(* Visualisation Lamp_status
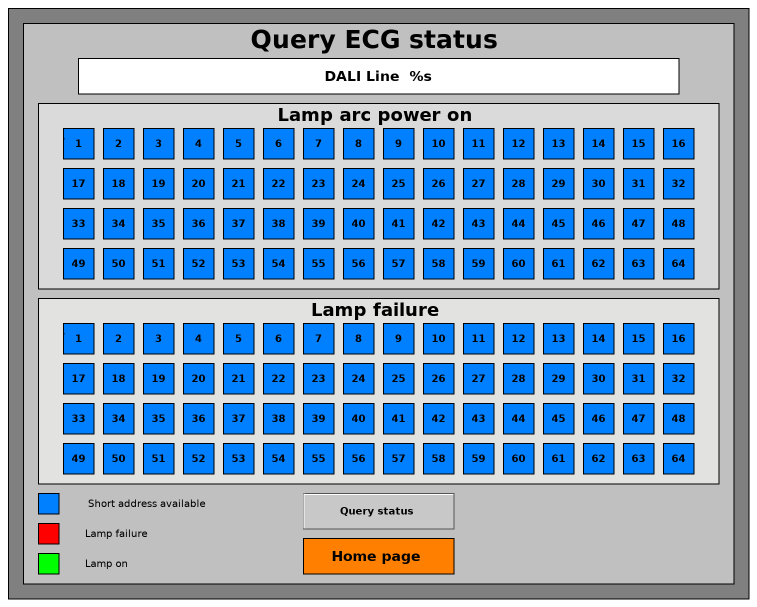
rectangle at (65,35)-(776,596): text "Query ECG status"
rounded rectangle at (345,550)-(496,586): text "Home page"; opens PLC_VISU; tooltip Back to home page
rounded rectangle at (120,70)-(721,106): text "DALI Line  %s"; shows DALI_Config.bDali_Linie; tooltip You can change the DALI Line only on the home page.
rectangle at (80,115)-(761,301): text "Lamp arc power on"
rectangle at (105,140)-(136,171): text "1"; alarm colour if DALI_Config.Kurzadr[1]
rectangle at (105,140)-(136,171): text "1"; invisible if not DALI_Config.Kurzadr[1]; alarm colour if DALI_Config.LampeEin[1]
rectangle at (145,140)-(176,171): text "2"; alarm colour if DALI_Config.Kurzadr[2]
rectangle at (145,140)-(176,171): text "2"; invisible if not DALI_Config.Kurzadr[2]; alarm colour if DALI_Config.LampeEin[2]
rectangle at (185,140)-(216,171): text "3"; alarm colour if DALI_Config.Kurzadr[3]
rectangle at (185,140)-(216,171): text "3"; invisible if not DALI_Config.Kurzadr[3]; alarm colour if DALI_Config.LampeEin[3]
rectangle at (225,140)-(256,171): text "4"; alarm colour if DALI_Config.Kurzadr[4]
rectangle at (225,140)-(256,171): text "4"; invisible if not DALI_Config.Kurzadr[4]; alarm colour if DALI_Config.LampeEin[4]
rectangle at (265,140)-(296,171): text "5"; alarm colour if DALI_Config.Kurzadr[5]
rectangle at (265,140)-(296,171): text "5"; invisible if not DALI_Config.Kurzadr[5]; alarm colour if DALI_Config.LampeEin[5]
rectangle at (305,140)-(336,171): text "6"; alarm colour if DALI_Config.Kurzadr[6]
rectangle at (305,140)-(336,171): text "6"; invisible if not DALI_Config.Kurzadr[6]; alarm colour if DALI_Config.LampeEin[6]
rectangle at (345,140)-(376,171): text "7"; alarm colour if DALI_Config.Kurzadr[7]
rectangle at (345,140)-(376,171): text "7"; invisible if not DALI_Config.Kurzadr[7]; alarm colour if DALI_Config.LampeEin[7]
rectangle at (385,140)-(416,171): text "8"; alarm colour if DALI_Config.Kurzadr[8]
rectangle at (385,140)-(416,171): text "8"; invisible if not DALI_Config.Kurzadr[8]; alarm colour if DALI_Config.LampeEin[8]
rectangle at (425,140)-(456,171): text "9"; alarm colour if DALI_Config.Kurzadr[9]
rectangle at (425,140)-(456,171): text "9"; invisible if not DALI_Config.Kurzadr[9]; alarm colour if DALI_Config.LampeEin[9]
rectangle at (465,140)-(496,171): text "10"; alarm colour if DALI_Config.Kurzadr[10]
rectangle at (465,140)-(496,171): text "10"; invisible if not DALI_Config.Kurzadr[10]; alarm colour if DALI_Config.LampeEin[10]
rectangle at (505,140)-(536,171): text "11"; alarm colour if DALI_Config.Kurzadr[11]
rectangle at (505,140)-(536,171): text "11"; invisible if not DALI_Config.Kurzadr[11]; alarm colour if DALI_Config.LampeEin[11]
rectangle at (545,140)-(576,171): text "12"; alarm colour if DALI_Config.Kurzadr[12]
rectangle at (545,140)-(576,171): text "12"; invisible if not DALI_Config.Kurzadr[12]; alarm colour if DALI_Config.LampeEin[12]
rectangle at (585,140)-(616,171): text "13"; alarm colour if DALI_Config.Kurzadr[13]
rectangle at (585,140)-(616,171): text "13"; invisible if not DALI_Config.Kurzadr[13]; alarm colour if DALI_Config.LampeEin[13]
rectangle at (625,140)-(656,171): text "14"; alarm colour if DALI_Config.Kurzadr[14]
rectangle at (625,140)-(656,171): text "14"; invisible if not DALI_Config.Kurzadr[14]; alarm colour if DALI_Config.LampeEin[14]
rectangle at (665,140)-(696,171): text "15"; alarm colour if DALI_Config.Kurzadr[15]
rectangle at (665,140)-(696,171): text "15"; invisible if not DALI_Config.Kurzadr[15]; alarm colour if DALI_Config.LampeEin[15]
rectangle at (705,140)-(736,171): text "16"; alarm colour if DALI_Config.Kurzadr[16]
rectangle at (705,140)-(736,171): text "16"; invisible if not DALI_Config.Kurzadr[16]; alarm colour if DALI_Config.LampeEin[16]
rectangle at (105,180)-(136,211): text "17"; alarm colour if DALI_Config.Kurzadr[17]
rectangle at (105,180)-(136,211): text "17"; invisible if not DALI_Config.Kurzadr[17]; alarm colour if DALI_Config.LampeEin[17]
rectangle at (185,180)-(216,211): text "19"; alarm colour if DALI_Config.Kurzadr[19]
rectangle at (185,180)-(216,211): text "19"; invisible if not DALI_Config.Kurzadr[19]; alarm colour if DALI_Config.LampeEin[19]
rectangle at (145,180)-(176,211): text "18"; alarm colour if DALI_Config.Kurzadr[18]
rectangle at (145,180)-(176,211): text "18"; invisible if not DALI_Config.Kurzadr[18]; alarm colour if DALI_Config.LampeEin[18]
rectangle at (225,180)-(256,211): text "20"; alarm colour if DALI_Config.Kurzadr[20]
rectangle at (225,180)-(256,211): text "20"; invisible if not DALI_Config.Kurzadr[20]; alarm colour if DALI_Config.LampeEin[20]
rectangle at (265,180)-(296,211): text "21"; alarm colour if DALI_Config.Kurzadr[21]
rectangle at (265,180)-(296,211): text "21"; invisible if not DALI_Config.Kurzadr[21]; alarm colour if DALI_Config.LampeEin[21]
rectangle at (305,180)-(336,211): text "22"; alarm colour if DALI_Config.Kurzadr[22]
rectangle at (305,180)-(336,211): text "22"; invisible if not DALI_Config.Kurzadr[22]; alarm colour if DALI_Config.LampeEin[22]
rectangle at (345,180)-(376,211): text "23"; alarm colour if DALI_Config.Kurzadr[23]
rectangle at (345,180)-(376,211): text "23"; invisible if not DALI_Config.Kurzadr[23]; alarm colour if DALI_Config.LampeEin[23]
rectangle at (385,180)-(416,211): text "24"; alarm colour if DALI_Config.Kurzadr[24]
rectangle at (385,180)-(416,211): text "24"; invisible if not DALI_Config.Kurzadr[24]; alarm colour if DALI_Config.LampeEin[24]
rectangle at (425,180)-(456,211): text "25"; alarm colour if DALI_Config.Kurzadr[25]
rectangle at (425,180)-(456,211): text "25"; invisible if not DALI_Config.Kurzadr[25]; alarm colour if DALI_Config.LampeEin[25]
rectangle at (585,180)-(616,211): text "29"; alarm colour if DALI_Config.Kurzadr[29]
rectangle at (585,180)-(616,211): text "29"; invisible if not DALI_Config.Kurzadr[29]; alarm colour if DALI_Config.LampeEin[29]
rectangle at (545,180)-(576,211): text "28"; alarm colour if DALI_Config.Kurzadr[28]
rectangle at (545,180)-(576,211): text "28"; invisible if not DALI_Config.Kurzadr[28]; alarm colour if DALI_Config.LampeEin[28]
rectangle at (505,180)-(536,211): text "27"; alarm colour if DALI_Config.Kurzadr[27]
rectangle at (505,180)-(536,211): text "27"; invisible if not DALI_Config.Kurzadr[27]; alarm colour if DALI_Config.LampeEin[27]
rectangle at (465,180)-(496,211): text "26"; alarm colour if DALI_Config.Kurzadr[26]
rectangle at (465,180)-(496,211): text "26"; invisible if not DALI_Config.Kurzadr[26]; alarm colour if DALI_Config.LampeEin[26]
rectangle at (625,180)-(656,211): text "30"; alarm colour if DALI_Config.Kurzadr[30]
rectangle at (625,180)-(656,211): text "30"; invisible if not DALI_Config.Kurzadr[30]; alarm colour if DALI_Config.LampeEin[30]
rectangle at (665,180)-(696,211): text "31"; alarm colour if DALI_Config.Kurzadr[31]
rectangle at (665,180)-(696,211): text "31"; invisible if not DALI_Config.Kurzadr[31]; alarm colour if DALI_Config.LampeEin[31]
rectangle at (705,180)-(736,211): text "32"; alarm colour if DALI_Config.Kurzadr[32]
rectangle at (705,180)-(736,211): text "32"; invisible if not DALI_Config.Kurzadr[32]; alarm colour if DALI_Config.LampeEin[32]
rectangle at (105,220)-(136,251): text "33"; alarm colour if DALI_Config.Kurzadr[33]
rectangle at (105,220)-(136,251): text "33"; invisible if not DALI_Config.Kurzadr[33]; alarm colour if DALI_Config.LampeEin[33]
rectangle at (145,220)-(176,251): text "34"; alarm colour if DALI_Config.Kurzadr[34]
rectangle at (145,220)-(176,251): text "34"; invisible if not DALI_Config.Kurzadr[34]; alarm colour if DALI_Config.LampeEin[34]
rectangle at (225,220)-(256,251): text "36"; alarm colour if DALI_Config.Kurzadr[36]
rectangle at (225,220)-(256,251): text "36"; invisible if not DALI_Config.Kurzadr[36]; alarm colour if DALI_Config.LampeEin[36]
rectangle at (305,220)-(336,251): text "38"; alarm colour if DALI_Config.Kurzadr[38]
rectangle at (305,220)-(336,251): text "38"; invisible if not DALI_Config.Kurzadr[38]; alarm colour if DALI_Config.LampeEin[38]
rectangle at (345,220)-(376,251): text "39"; alarm colour if DALI_Config.Kurzadr[39]
rectangle at (345,220)-(376,251): text "39"; invisible if not DALI_Config.Kurzadr[39]; alarm colour if DALI_Config.LampeEin[39]
rectangle at (265,220)-(296,251): text "37"; alarm colour if DALI_Config.Kurzadr[37]
rectangle at (265,220)-(296,251): text "37"; invisible if not DALI_Config.Kurzadr[37]; alarm colour if DALI_Config.LampeEin[37]
rectangle at (185,220)-(216,251): text "35"; alarm colour if DALI_Config.Kurzadr[35]
rectangle at (185,220)-(216,251): text "35"; invisible if not DALI_Config.Kurzadr[35]; alarm colour if DALI_Config.LampeEin[35]
rectangle at (425,220)-(456,251): text "41"; alarm colour if DALI_Config.Kurzadr[41]
rectangle at (425,220)-(456,251): text "41"; invisible if not DALI_Config.Kurzadr[41]; alarm colour if DALI_Config.LampeEin[41]
rectangle at (465,220)-(496,251): text "42"; alarm colour if DALI_Config.Kurzadr[42]
rectangle at (465,220)-(496,251): text "42"; invisible if not DALI_Config.Kurzadr[42]; alarm colour if DALI_Config.LampeEin[42]
rectangle at (385,220)-(416,251): text "40"; alarm colour if DALI_Config.Kurzadr[40]
rectangle at (385,220)-(416,251): text "40"; invisible if not DALI_Config.Kurzadr[40]; alarm colour if DALI_Config.LampeEin[40]
rectangle at (505,220)-(536,251): text "43"; alarm colour if DALI_Config.Kurzadr[43]
rectangle at (505,220)-(536,251): text "43"; invisible if not DALI_Config.Kurzadr[43]; alarm colour if DALI_Config.LampeEin[43]
rectangle at (545,220)-(576,251): text "44"; alarm colour if DALI_Config.Kurzadr[44]
rectangle at (545,220)-(576,251): text "44"; invisible if not DALI_Config.Kurzadr[44]; alarm colour if DALI_Config.LampeEin[44]
rectangle at (585,220)-(616,251): text "45"; alarm colour if DALI_Config.Kurzadr[45]
rectangle at (585,220)-(616,251): text "45"; invisible if not DALI_Config.Kurzadr[45]; alarm colour if DALI_Config.LampeEin[45]
rectangle at (625,220)-(656,251): text "46"; alarm colour if DALI_Config.Kurzadr[46]
rectangle at (625,220)-(656,251): text "46"; invisible if not DALI_Config.Kurzadr[46]; alarm colour if DALI_Config.LampeEin[46]
rectangle at (665,220)-(696,251): text "47"; alarm colour if DALI_Config.Kurzadr[47]
rectangle at (665,220)-(696,251): text "47"; invisible if not DALI_Config.Kurzadr[47]; alarm colour if DALI_Config.LampeEin[47]
rectangle at (705,220)-(736,251): text "48"; alarm colour if DALI_Config.Kurzadr[48]
rectangle at (705,220)-(736,251): text "48"; invisible if not DALI_Config.Kurzadr[48]; alarm colour if DALI_Config.LampeEin[48]
rectangle at (105,260)-(136,291): text "49"; alarm colour if DALI_Config.Kurzadr[49]
rectangle at (105,260)-(136,291): text "49"; invisible if not DALI_Config.Kurzadr[49]; alarm colour if DALI_Config.LampeEin[49]
rectangle at (145,260)-(176,291): text "50"; alarm colour if DALI_Config.Kurzadr[50]
rectangle at (145,260)-(176,291): text "50"; invisible if not DALI_Config.Kurzadr[50]; alarm colour if DALI_Config.LampeEin[50]
rectangle at (185,260)-(216,291): text "51"; alarm colour if DALI_Config.Kurzadr[51]
rectangle at (185,260)-(216,291): text "51"; invisible if not DALI_Config.Kurzadr[51]; alarm colour if DALI_Config.LampeEin[51]
rectangle at (225,260)-(256,291): text "52"; alarm colour if DALI_Config.Kurzadr[52]
rectangle at (225,260)-(256,291): text "52"; invisible if not DALI_Config.Kurzadr[52]; alarm colour if DALI_Config.LampeEin[52]
rectangle at (265,260)-(296,291): text "53"; alarm colour if DALI_Config.Kurzadr[53]
rectangle at (265,260)-(296,291): text "53"; invisible if not DALI_Config.Kurzadr[53]; alarm colour if DALI_Config.LampeEin[53]
rectangle at (305,260)-(336,291): text "54"; alarm colour if DALI_Config.Kurzadr[54]
rectangle at (305,260)-(336,291): text "54"; invisible if not DALI_Config.Kurzadr[54]; alarm colour if DALI_Config.LampeEin[54]
rectangle at (345,260)-(376,291): text "55"; alarm colour if DALI_Config.Kurzadr[55]
rectangle at (345,260)-(376,291): text "55"; invisible if not DALI_Config.Kurzadr[55]; alarm colour if DALI_Config.LampeEin[55]
rectangle at (385,260)-(416,291): text "56"; alarm colour if DALI_Config.Kurzadr[56]
rectangle at (385,260)-(416,291): text "56"; invisible if not DALI_Config.Kurzadr[56]; alarm colour if DALI_Config.LampeEin[56]
rectangle at (425,260)-(456,291): text "57"; alarm colour if DALI_Config.Kurzadr[57]
rectangle at (425,260)-(456,291): text "57"; invisible if not DALI_Config.Kurzadr[57]; alarm colour if DALI_Config.LampeEin[57]
rectangle at (505,260)-(536,291): text "59"; alarm colour if DALI_Config.Kurzadr[59]
rectangle at (505,260)-(536,291): text "59"; invisible if not DALI_Config.Kurzadr[59]; alarm colour if DALI_Config.LampeEin[59]
rectangle at (545,260)-(576,291): text "60"; alarm colour if DALI_Config.Kurzadr[60]
rectangle at (545,260)-(576,291): text "60"; invisible if not DALI_Config.Kurzadr[60]; alarm colour if DALI_Config.LampeEin[60]
rectangle at (585,260)-(616,291): text "61"; alarm colour if DALI_Config.Kurzadr[61]
rectangle at (585,260)-(616,291): text "61"; invisible if not DALI_Config.Kurzadr[61]; alarm colour if DALI_Config.LampeEin[61]
rectangle at (625,260)-(656,291): text "62"; alarm colour if DALI_Config.Kurzadr[62]
rectangle at (625,260)-(656,291): text "62"; invisible if not DALI_Config.Kurzadr[62]; alarm colour if DALI_Config.LampeEin[62]
rectangle at (465,260)-(496,291): text "58"; alarm colour if DALI_Config.Kurzadr[58]
rectangle at (465,260)-(496,291): text "58"; invisible if not DALI_Config.Kurzadr[58]; alarm colour if DALI_Config.LampeEin[58]
rectangle at (665,260)-(696,291): text "63"; alarm colour if DALI_Config.Kurzadr[63]
rectangle at (665,260)-(696,291): text "63"; invisible if not DALI_Config.Kurzadr[63]; alarm colour if DALI_Config.LampeEin[63]
rectangle at (705,260)-(736,291): text "64"; alarm colour if DALI_Config.Kurzadr[64]
rectangle at (705,260)-(736,291): text "64"; invisible if not DALI_Config.Kurzadr[64]; alarm colour if DALI_Config.LampeEin[64]
rectangle at (80,310)-(761,496): text "Lamp failure"
rectangle at (105,335)-(136,366): text "1"; alarm colour if DALI_Config.Kurzadr[1]
rectangle at (105,335)-(136,366): text "1"; invisible if not DALI_Config.Kurzadr[1]; alarm colour if DALI_Config.Lampenausfall[1]
rectangle at (145,335)-(176,366): text "2"; alarm colour if DALI_Config.Kurzadr[2]
rectangle at (145,335)-(176,366): text "2"; invisible if not DALI_Config.Kurzadr[2]; alarm colour if DALI_Config.Lampenausfall[2]
rectangle at (185,335)-(216,366): text "3"; alarm colour if DALI_Config.Kurzadr[3]
rectangle at (185,335)-(216,366): text "3"; invisible if not DALI_Config.Kurzadr[3]; alarm colour if DALI_Config.Lampenausfall[3]
rectangle at (225,335)-(256,366): text "4"; alarm colour if DALI_Config.Kurzadr[4]
rectangle at (225,335)-(256,366): text "4"; invisible if not DALI_Config.Kurzadr[4]; alarm colour if DALI_Config.Lampenausfall[4]
rectangle at (265,335)-(296,366): text "5"; alarm colour if DALI_Config.Kurzadr[5]
rectangle at (265,335)-(296,366): text "5"; invisible if not DALI_Config.Kurzadr[5]; alarm colour if DALI_Config.Lampenausfall[5]
rectangle at (305,335)-(336,366): text "6"; alarm colour if DALI_Config.Kurzadr[6]
rectangle at (305,335)-(336,366): text "6"; invisible if not DALI_Config.Kurzadr[6]; alarm colour if DALI_Config.Lampenausfall[6]
rectangle at (345,335)-(376,366): text "7"; alarm colour if DALI_Config.Kurzadr[7]
rectangle at (345,335)-(376,366): text "7"; invisible if not DALI_Config.Kurzadr[7]; alarm colour if DALI_Config.Lampenausfall[7]
rectangle at (385,335)-(416,366): text "8"; alarm colour if DALI_Config.Kurzadr[8]
rectangle at (385,335)-(416,366): text "8"; invisible if not DALI_Config.Kurzadr[8]; alarm colour if DALI_Config.Lampenausfall[8]
rectangle at (425,335)-(456,366): text "9"; alarm colour if DALI_Config.Kurzadr[9]
rectangle at (425,335)-(456,366): text "9"; invisible if not DALI_Config.Kurzadr[9]; alarm colour if DALI_Config.Lampenausfall[9]
rectangle at (465,335)-(496,366): text "10"; alarm colour if DALI_Config.Kurzadr[10]
rectangle at (465,335)-(496,366): text "10"; invisible if not DALI_Config.Kurzadr[10]; alarm colour if DALI_Config.Lampenausfall[10]
rectangle at (505,335)-(536,366): text "11"; alarm colour if DALI_Config.Kurzadr[11]
rectangle at (505,335)-(536,366): text "11"; invisible if not DALI_Config.Kurzadr[11]; alarm colour if DALI_Config.Lampenausfall[11]
rectangle at (545,335)-(576,366): text "12"; alarm colour if DALI_Config.Kurzadr[12]
rectangle at (545,335)-(576,366): text "12"; invisible if not DALI_Config.Kurzadr[12]; alarm colour if DALI_Config.Lampenausfall[12]
rectangle at (585,335)-(616,366): text "13"; alarm colour if DALI_Config.Kurzadr[13]
rectangle at (585,335)-(616,366): text "13"; invisible if not DALI_Config.Kurzadr[13]; alarm colour if DALI_Config.Lampenausfall[13]
rectangle at (625,335)-(656,366): text "14"; alarm colour if DALI_Config.Kurzadr[14]
rectangle at (625,335)-(656,366): text "14"; invisible if not DALI_Config.Kurzadr[14]; alarm colour if DALI_Config.Lampenausfall[14]
rectangle at (665,335)-(696,366): text "15"; alarm colour if DALI_Config.Kurzadr[15]
rectangle at (665,335)-(696,366): text "15"; invisible if not DALI_Config.Kurzadr[15]; alarm colour if DALI_Config.Lampenausfall[15]
rectangle at (705,335)-(736,366): text "16"; alarm colour if DALI_Config.Kurzadr[16]
rectangle at (705,335)-(736,366): text "16"; invisible if not DALI_Config.Kurzadr[16]; alarm colour if DALI_Config.Lampenausfall[16]
rectangle at (105,375)-(136,406): text "17"; alarm colour if DALI_Config.Kurzadr[17]
rectangle at (105,375)-(136,406): text "17"; invisible if not DALI_Config.Kurzadr[17]; alarm colour if DALI_Config.Lampenausfall[17]
rectangle at (185,375)-(216,406): text "19"; alarm colour if DALI_Config.Kurzadr[19]
rectangle at (185,375)-(216,406): text "19"; invisible if not DALI_Config.Kurzadr[19]; alarm colour if DALI_Config.Lampenausfall[19]
rectangle at (145,375)-(176,406): text "18"; alarm colour if DALI_Config.Kurzadr[18]
rectangle at (145,375)-(176,406): text "18"; invisible if not DALI_Config.Kurzadr[18]; alarm colour if DALI_Config.Lampenausfall[18]
rectangle at (225,375)-(256,406): text "20"; alarm colour if DALI_Config.Kurzadr[20]
rectangle at (225,375)-(256,406): text "20"; invisible if not DALI_Config.Kurzadr[20]; alarm colour if DALI_Config.Lampenausfall[20]
rectangle at (265,375)-(296,406): text "21"; alarm colour if DALI_Config.Kurzadr[21]
rectangle at (265,375)-(296,406): text "21"; invisible if not DALI_Config.Kurzadr[21]; alarm colour if DALI_Config.Lampenausfall[21]
rectangle at (305,375)-(336,406): text "22"; alarm colour if DALI_Config.Kurzadr[22]
rectangle at (305,375)-(336,406): text "22"; invisible if not DALI_Config.Kurzadr[22]; alarm colour if DALI_Config.Lampenausfall[22]
rectangle at (345,375)-(376,406): text "23"; alarm colour if DALI_Config.Kurzadr[23]
rectangle at (345,375)-(376,406): text "23"; invisible if not DALI_Config.Kurzadr[23]; alarm colour if DALI_Config.Lampenausfall[23]
rectangle at (385,375)-(416,406): text "24"; alarm colour if DALI_Config.Kurzadr[24]
rectangle at (385,375)-(416,406): text "24"; invisible if not DALI_Config.Kurzadr[24]; alarm colour if DALI_Config.Lampenausfall[24]
rectangle at (425,375)-(456,406): text "25"; alarm colour if DALI_Config.Kurzadr[25]
rectangle at (425,375)-(456,406): text "25"; invisible if not DALI_Config.Kurzadr[25]; alarm colour if DALI_Config.Lampenausfall[25]
rectangle at (585,375)-(616,406): text "29"; alarm colour if DALI_Config.Kurzadr[29]
rectangle at (585,375)-(616,406): text "29"; invisible if not DALI_Config.Kurzadr[29]; alarm colour if DALI_Config.Lampenausfall[29]
rectangle at (545,375)-(576,406): text "28"; alarm colour if DALI_Config.Kurzadr[28]
rectangle at (545,375)-(576,406): text "28"; invisible if not DALI_Config.Kurzadr[28]; alarm colour if DALI_Config.Lampenausfall[28]
rectangle at (505,375)-(536,406): text "27"; alarm colour if DALI_Config.Kurzadr[27]
rectangle at (505,375)-(536,406): text "27"; invisible if not DALI_Config.Kurzadr[27]; alarm colour if DALI_Config.Lampenausfall[27]
rectangle at (465,375)-(496,406): text "26"; alarm colour if DALI_Config.Kurzadr[26]
rectangle at (465,375)-(496,406): text "26"; invisible if not DALI_Config.Kurzadr[26]; alarm colour if DALI_Config.Lampenausfall[26]
rectangle at (625,375)-(656,406): text "30"; alarm colour if DALI_Config.Kurzadr[30]
rectangle at (625,375)-(656,406): text "30"; invisible if not DALI_Config.Kurzadr[30]; alarm colour if DALI_Config.Lampenausfall[30]
rectangle at (665,375)-(696,406): text "31"; alarm colour if DALI_Config.Kurzadr[31]
rectangle at (665,375)-(696,406): text "31"; invisible if not DALI_Config.Kurzadr[31]; alarm colour if DALI_Config.Lampenausfall[31]
rectangle at (705,375)-(736,406): text "32"; alarm colour if DALI_Config.Kurzadr[32]
rectangle at (705,375)-(736,406): text "32"; invisible if not DALI_Config.Kurzadr[32]; alarm colour if DALI_Config.Lampenausfall[32]
rectangle at (105,415)-(136,446): text "33"; alarm colour if DALI_Config.Kurzadr[33]
rectangle at (105,415)-(136,446): text "33"; invisible if not DALI_Config.Kurzadr[33]; alarm colour if DALI_Config.Lampenausfall[33]
rectangle at (145,415)-(176,446): text "34"; alarm colour if DALI_Config.Kurzadr[34]
rectangle at (145,415)-(176,446): text "34"; invisible if not DALI_Config.Kurzadr[34]; alarm colour if DALI_Config.Lampenausfall[34]
rectangle at (225,415)-(256,446): text "36"; alarm colour if DALI_Config.Kurzadr[36]
rectangle at (225,415)-(256,446): text "36"; invisible if not DALI_Config.Kurzadr[36]; alarm colour if DALI_Config.Lampenausfall[36]
rectangle at (305,415)-(336,446): text "38"; alarm colour if DALI_Config.Kurzadr[38]
rectangle at (305,415)-(336,446): text "38"; invisible if not DALI_Config.Kurzadr[38]; alarm colour if DALI_Config.Lampenausfall[38]
rectangle at (345,415)-(376,446): text "39"; alarm colour if DALI_Config.Kurzadr[39]
rectangle at (345,415)-(376,446): text "39"; invisible if not DALI_Config.Kurzadr[39]; alarm colour if DALI_Config.Lampenausfall[39]
rectangle at (265,415)-(296,446): text "37"; alarm colour if DALI_Config.Kurzadr[37]
rectangle at (265,415)-(296,446): text "37"; invisible if not DALI_Config.Kurzadr[37]; alarm colour if DALI_Config.Lampenausfall[37]
rectangle at (185,415)-(216,446): text "35"; alarm colour if DALI_Config.Kurzadr[35]
rectangle at (185,415)-(216,446): text "35"; invisible if not DALI_Config.Kurzadr[35]; alarm colour if DALI_Config.Lampenausfall[35]
rectangle at (425,415)-(456,446): text "41"; alarm colour if DALI_Config.Kurzadr[41]
rectangle at (425,415)-(456,446): text "41"; invisible if not DALI_Config.Kurzadr[41]; alarm colour if DALI_Config.Lampenausfall[41]
rectangle at (465,415)-(496,446): text "42"; alarm colour if DALI_Config.Kurzadr[42]
rectangle at (465,415)-(496,446): text "42"; invisible if not DALI_Config.Kurzadr[42]; alarm colour if DALI_Config.Lampenausfall[42]
rectangle at (385,415)-(416,446): text "40"; alarm colour if DALI_Config.Kurzadr[40]
rectangle at (385,415)-(416,446): text "40"; invisible if not DALI_Config.Kurzadr[40]; alarm colour if DALI_Config.Lampenausfall[40]
rectangle at (505,415)-(536,446): text "43"; alarm colour if DALI_Config.Kurzadr[43]
rectangle at (505,415)-(536,446): text "43"; invisible if not DALI_Config.Kurzadr[43]; alarm colour if DALI_Config.Lampenausfall[43]
rectangle at (545,415)-(576,446): text "44"; alarm colour if DALI_Config.Kurzadr[44]
rectangle at (545,415)-(576,446): text "44"; invisible if not DALI_Config.Kurzadr[44]; alarm colour if DALI_Config.Lampenausfall[44]
rectangle at (585,415)-(616,446): text "45"; alarm colour if DALI_Config.Kurzadr[45]
rectangle at (585,415)-(616,446): text "45"; invisible if not DALI_Config.Kurzadr[45]; alarm colour if DALI_Config.Lampenausfall[45]
rectangle at (625,415)-(656,446): text "46"; alarm colour if DALI_Config.Kurzadr[46]
rectangle at (625,415)-(656,446): text "46"; invisible if not DALI_Config.Kurzadr[46]; alarm colour if DALI_Config.Lampenausfall[46]
rectangle at (665,415)-(696,446): text "47"; alarm colour if DALI_Config.Kurzadr[47]
rectangle at (665,415)-(696,446): text "47"; invisible if not DALI_Config.Kurzadr[47]; alarm colour if DALI_Config.Lampenausfall[47]
rectangle at (705,415)-(736,446): text "48"; alarm colour if DALI_Config.Kurzadr[48]
rectangle at (705,415)-(736,446): text "48"; invisible if not DALI_Config.Kurzadr[48]; alarm colour if DALI_Config.Lampenausfall[48]
rectangle at (105,455)-(136,486): text "49"; alarm colour if DALI_Config.Kurzadr[49]
rectangle at (105,455)-(136,486): text "49"; invisible if not DALI_Config.Kurzadr[49]; alarm colour if DALI_Config.Lampenausfall[49]
rectangle at (145,455)-(176,486): text "50"; alarm colour if DALI_Config.Kurzadr[50]
rectangle at (145,455)-(176,486): text "50"; invisible if not DALI_Config.Kurzadr[50]; alarm colour if DALI_Config.Lampenausfall[50]
rectangle at (185,455)-(216,486): text "51"; alarm colour if DALI_Config.Kurzadr[51]
rectangle at (185,455)-(216,486): text "51"; invisible if not DALI_Config.Kurzadr[51]; alarm colour if DALI_Config.Lampenausfall[51]
rectangle at (225,455)-(256,486): text "52"; alarm colour if DALI_Config.Kurzadr[52]
rectangle at (225,455)-(256,486): text "52"; invisible if not DALI_Config.Kurzadr[52]; alarm colour if DALI_Config.Lampenausfall[52]
rectangle at (265,455)-(296,486): text "53"; alarm colour if DALI_Config.Kurzadr[53]
rectangle at (265,455)-(296,486): text "53"; invisible if not DALI_Config.Kurzadr[53]; alarm colour if DALI_Config.Lampenausfall[53]
rectangle at (305,455)-(336,486): text "54"; alarm colour if DALI_Config.Kurzadr[54]
rectangle at (305,455)-(336,486): text "54"; invisible if not DALI_Config.Kurzadr[54]; alarm colour if DALI_Config.Lampenausfall[54]
rectangle at (345,455)-(376,486): text "55"; alarm colour if DALI_Config.Kurzadr[55]
rectangle at (345,455)-(376,486): text "55"; invisible if not DALI_Config.Kurzadr[55]; alarm colour if DALI_Config.Lampenausfall[55]
rectangle at (385,455)-(416,486): text "56"; alarm colour if DALI_Config.Kurzadr[56]
rectangle at (385,455)-(416,486): text "56"; invisible if not DALI_Config.Kurzadr[56]; alarm colour if DALI_Config.Lampenausfall[56]
rectangle at (425,455)-(456,486): text "57"; alarm colour if DALI_Config.Kurzadr[57]
rectangle at (425,455)-(456,486): text "57"; invisible if not DALI_Config.Kurzadr[57]; alarm colour if DALI_Config.Lampenausfall[57]
rectangle at (505,455)-(536,486): text "59"; alarm colour if DALI_Config.Kurzadr[59]
rectangle at (505,455)-(536,486): text "59"; invisible if not DALI_Config.Kurzadr[59]; alarm colour if DALI_Config.Lampenausfall[59]
rectangle at (545,455)-(576,486): text "60"; alarm colour if DALI_Config.Kurzadr[60]
rectangle at (545,455)-(576,486): text "60"; invisible if not DALI_Config.Kurzadr[60]; alarm colour if DALI_Config.Lampenausfall[60]
rectangle at (585,455)-(616,486): text "61"; alarm colour if DALI_Config.Kurzadr[61]
rectangle at (585,455)-(616,486): text "61"; invisible if not DALI_Config.Kurzadr[61]; alarm colour if DALI_Config.Lampenausfall[61]
rectangle at (625,455)-(656,486): text "62"; alarm colour if DALI_Config.Kurzadr[62]
rectangle at (625,455)-(656,486): text "62"; invisible if not DALI_Config.Kurzadr[62]; alarm colour if DALI_Config.Lampenausfall[62]
rectangle at (465,455)-(496,486): text "58"; alarm colour if DALI_Config.Kurzadr[58]
rectangle at (465,455)-(496,486): text "58"; invisible if not DALI_Config.Kurzadr[58]; alarm colour if DALI_Config.Lampenausfall[58]
rectangle at (665,455)-(696,486): text "63"; alarm colour if DALI_Config.Kurzadr[63]
rectangle at (665,455)-(696,486): text "63"; invisible if not DALI_Config.Kurzadr[63]; alarm colour if DALI_Config.Lampenausfall[63]
rectangle at (705,455)-(736,486): text "64"; alarm colour if DALI_Config.Kurzadr[64]
rectangle at (705,455)-(736,486): text "64"; invisible if not DALI_Config.Kurzadr[64]; alarm colour if DALI_Config.Lampenausfall[64]
button at (345,505)-(496,541): text "Query status"; taps DALI_Config.Status; tooltip If you click the button "Query Status", you will get the status "Lamp failure" and "Lamp arc power on" from the ECG.
rectangle at (110,505)-(271,526): text "Short address available"
rectangle at (125,535)-(256,556): text "Lamp failure"
rectangle at (125,565)-(196,586): text "Lamp on"
6 more shapes without text or variables
*)

(* Visualisation lux
rectangle at (915,525)-(1011,546): text "Zpet"; opens PLC_VISU; tooltip Back to home page
1 elements of other kinds (tables, trends, ...) not read
*)

(* Visualisation PLC_VISU
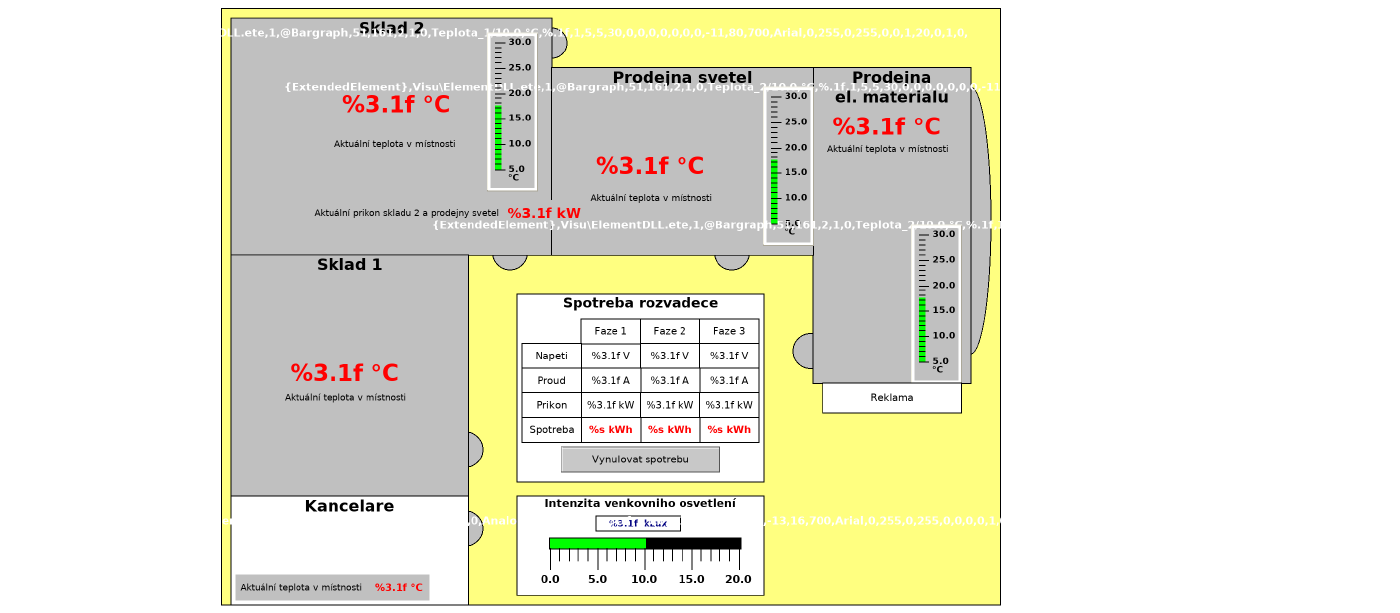
ellipse at (740,80)-(781,351): opens CasProg
ellipse at (580,330)-(616,366): alarm colour if .KA13; taps .TL10s; tooltip Dlouhý stisk zapne svìtlo. (cca 1s)
rectangle at (600,60)-(761,381): text "Prodejna"; opens prodej_materialu
ellipse at (500,230)-(536,266): alarm colour if .KA13; taps .TL10s; tooltip Dlouhý stisk zapne svìtlo. (cca 1s)
ellipse at (275,230)-(311,266): alarm colour if .KA16; taps .TL05s; tooltip Dlouhý stisk zapne svìtlo. (cca 1s)
ellipse at (320,20)-(351,51): alarm colour if .KA15; taps .TL06s; tooltip Dlouhý stisk zapne svìtlo. (cca 1s)
rectangle at (10,10)-(336,251): text "Sklad 2"; opens DALI_cfg
rectangle at (10,250)-(251,496): text "Sklad 1"; opens DALI_cfg
rectangle at (335,60)-(601,251): text "Prodejna svetel"; opens prodej_svetel
rectangle at (10,495)-(251,606): text "Kancelare"
rectangle at (60,380)-(201,411): text "Aktuální teplota v místnosti"
rectangle at (70,350)-(181,391): text "%3.1f °C"; shows .Teplota_3/10.0
rectangle at (110,125)-(251,151): text "Aktuální teplota v místnosti"
rectangle at (120,70)-(236,126): text "%3.1f °C"; shows .Teplota_1/10.0
rectangle at (380,130)-(491,191): text "%3.1f °C"; shows .Teplota_2/10.0
rectangle at (370,180)-(506,206): text "Aktuální teplota v místnosti"
rectangle at (15,575)-(151,601): text "Aktuální teplota v místnosti"
rectangle at (150,575)-(211,601): text "%3.1f °C"; shows .Teplota_4/10.0
rounded rectangle at (300,290)-(551,481): text "Spotreba rozvadece"
rectangle at (365,340)-(426,366): text "%3.1f V"; shows TriFaze.arNapeti[1]
rectangle at (365,315)-(426,341): text "Faze 1"
rectangle at (425,315)-(486,341): text "Faze 2"
rectangle at (485,315)-(546,341): text "Faze 3"
rectangle at (425,340)-(486,366): text "%3.1f V"; shows TriFaze.arNapeti[2]
rectangle at (485,340)-(546,366): text "%3.1f V"; shows TriFaze.arNapeti[3]
rectangle at (485,365)-(546,391): text "%3.1f A"; shows TriFaze.arProud[3]
rectangle at (425,365)-(486,391): text "%3.1f A"; shows TriFaze.arProud[2]
rectangle at (365,365)-(426,391): text "%3.1f A"; shows TriFaze.arProud[1]
rectangle at (365,390)-(426,416): text "%3.1f kW"; shows TriFaze.arVykon[1]
rectangle at (425,390)-(486,416): text "%3.1f kW"; shows TriFaze.arVykon[2]
rectangle at (485,390)-(546,416): text "%3.1f kW"; shows TriFaze.arVykon[3]
rectangle at (485,415)-(546,441): text "%s kWh"; shows TriFaze.adwSpotreba[3]
rectangle at (425,415)-(486,441): text "%s kWh"; shows TriFaze.adwSpotreba[2]
rectangle at (365,415)-(426,441): text "%s kWh"; shows TriFaze.adwSpotreba[1]
button at (345,445)-(506,471): text "Vynulovat spotrebu"; taps TriFaze.SmazL1
rounded rectangle at (300,495)-(551,596): text "Intenzita venkovniho osvetlení"; opens lux
rectangle at (380,515)-(466,531): text "%3.1f  kLux"; shows .Analog_1/3276.4*2
rectangle at (305,340)-(366,366): text "Napeti"
rectangle at (305,365)-(366,391): text "Proud"
rectangle at (305,390)-(366,416): text "Prikon"
rectangle at (305,415)-(366,441): text "Spotreba"
rectangle at (90,195)-(301,221): text "Aktuální prikon skladu 2 a prodejny svetel"
rectangle at (295,195)-(361,221): text "%3.1f kW"; shows TriFaze.arVykon[1]+TriFaze.arVykon[2]+TriFaze.arVykon[3]
group at (320,520)-(541,621)
  rectangle at (0,0)-(1,1): text "{ExtendedElement},Visu\ElementDLL.ete,1,@Bargraph,221,111,0,0,0,Analog_1/3276.4*2,,%.1f,1,5,0,20,0,0,0,0,0,0,0,-13,16,700,Arial,0,255,0,255,0,0,0,0,1,0,0,"
  rectangle at (14,19)-(111,29): alarm colour if (Analog_1/3276.4*2) < 0; right ((Analog_1/3276.4*2 * 1.0) - 10)  * 9.6
  rectangle at (2,53)-(26,103): text "0.0"
  rectangle at (50,53)-(74,103): text "5.0"
  rectangle at (93,53)-(126,103): text "10.0"
  rectangle at (141,53)-(174,103): text "15.0"
  rectangle at (189,53)-(222,103): text "20.0"
group at (550,80)-(601,241)
  rectangle at (0,0)-(1,1): text "{ExtendedElement},Visu\ElementDLL.ete,1,@Bargraph,51,161,2,1,0,Teplota_2/10.0,°C,%.1f,1,5,5,30,0,0,0,0,0,0,0,-11,80,700,Arial,0,255,0,255,0,0,1,25,0,1,0,"
  rectangle at (8,74)-(14,139): alarm colour if (Teplota_2/10.0) > 25; top ((Teplota_2/10.0 * 1.0) - 17.5)  * -5.2
  rectangle at (20,129)-(47,148): text "5.0"
  rectangle at (20,103)-(47,122): text "10.0"
  rectangle at (20,77)-(47,96): text "15.0"
  rectangle at (20,52)-(47,71): text "20.0"
  rectangle at (20,26)-(47,45): text "25.0"
  rectangle at (20,0)-(47,19): text "30.0"
  rectangle at (15,140)-(39,154): text "°C"
group at (270,25)-(321,186)
  rectangle at (0,0)-(1,1): text "{ExtendedElement},Visu\ElementDLL.ete,1,@Bargraph,51,161,2,1,0,Teplota_1/10.0,°C,%.1f,1,5,5,30,0,0,0,0,0,0,0,-11,80,700,Arial,0,255,0,255,0,0,1,20,0,1,0,"
  rectangle at (8,74)-(14,139): alarm colour if (Teplota_1/10.0) > 20; top ((Teplota_1/10.0 * 1.0) - 17.5)  * -5.2
  rectangle at (20,129)-(47,148): text "5.0"
  rectangle at (20,103)-(47,122): text "10.0"
  rectangle at (20,77)-(47,96): text "15.0"
  rectangle at (20,52)-(47,71): text "20.0"
  rectangle at (20,26)-(47,45): text "25.0"
  rectangle at (20,0)-(47,19): text "30.0"
  rectangle at (15,140)-(39,154): text "°C"
group at (700,220)-(751,381)
  rectangle at (0,0)-(1,1): text "{ExtendedElement},Visu\ElementDLL.ete,1,@Bargraph,51,161,2,1,0,Teplota_2/10.0,°C,%.1f,1,5,5,30,0,0,0,0,0,0,0,-11,80,700,Arial,0,255,0,255,0,0,1,25,0,1,0,"
  rectangle at (8,74)-(14,139): alarm colour if (Teplota_2/10.0) > 25; top ((Teplota_2/10.0 * 1.0) - 17.5)  * -5.2
  rectangle at (20,129)-(47,148): text "5.0"
  rectangle at (20,103)-(47,122): text "10.0"
  rectangle at (20,77)-(47,96): text "15.0"
  rectangle at (20,52)-(47,71): text "20.0"
  rectangle at (20,26)-(47,45): text "25.0"
  rectangle at (20,0)-(47,19): text "30.0"
  rectangle at (15,140)-(39,154): text "°C"
rectangle at (620,90)-(731,151): text "%3.1f °C"
rectangle at (610,130)-(746,156): text "Aktuální teplota v místnosti"
rectangle at (620,80)-(741,101): text "el. materialu"; opens prodej_materialu
rectangle at (610,380)-(751,411): text "Reklama"; opens CasProg
127 more shapes without text or variables
*)

(* Visualisation prodej_materialu
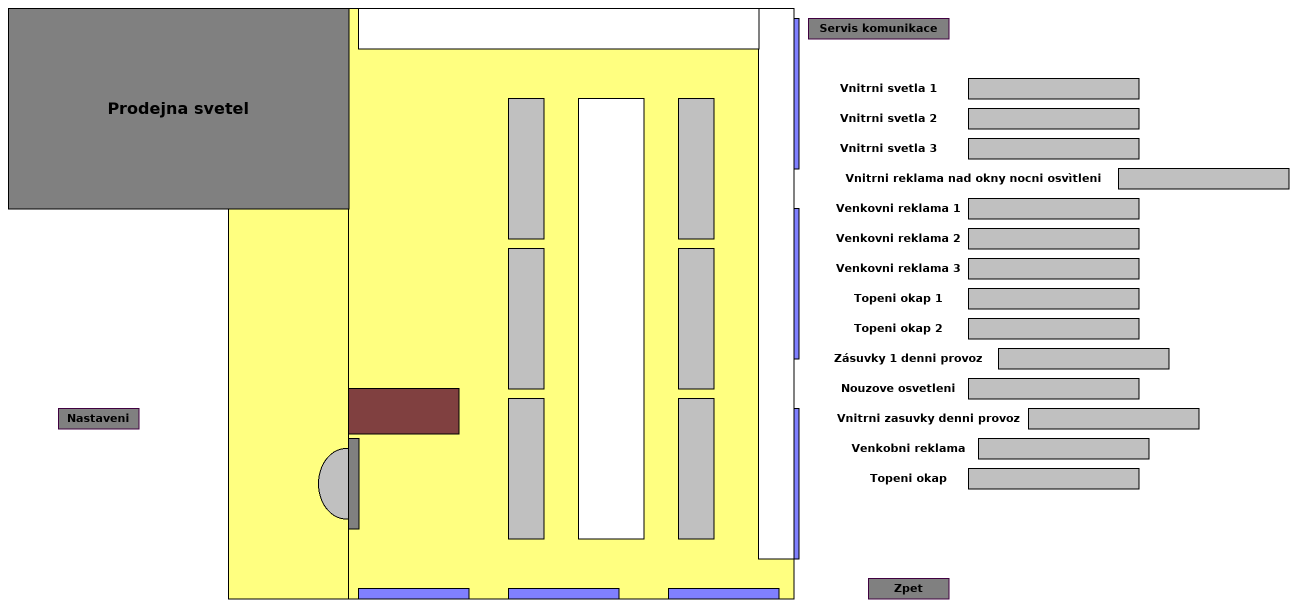
ellipse at (310,440)-(366,511): alarm colour if OUTSvetloNadVchodem; taps INSvetloNadVchodem; tooltip Dlouhý stisk zapne svìtlo. (cca 1s)
rectangle at (860,570)-(941,591): text "Zpet"; opens PLC_VISU; tooltip Back to home page
rectangle at (670,90)-(706,231): tooltip Kliknutím zapínáte a vypínáte svìtla DALI
rectangle at (670,240)-(706,381): tooltip Kliknutím zapínáte a vypínáte svìtla DALI
rectangle at (670,390)-(706,531): tooltip Kliknutím zapínáte a vypínáte svìtla DALI
rectangle at (500,90)-(536,231): tooltip Kliknutím zapínáte a vypínáte svìtla DALI
rectangle at (500,240)-(536,381): tooltip Kliknutím zapínáte a vypínáte svìtla DALI
rectangle at (500,390)-(536,531): tooltip Kliknutím zapínáte a vypínáte svìtla DALI
rectangle at (0,0)-(341,201): text "Prodejna svetel"; opens prodej_svetel
rectangle at (750,0)-(786,551): tooltip Kliknutím zapínáte a vypínáte svìtla DALI
rectangle at (570,90)-(636,531): tooltip Kliknutím zapínáte a vypínáte svìtla DALI
rectangle at (350,0)-(751,41): tooltip Kliknutím zapínáte a vypínáte svìtla DALI
rectangle at (800,10)-(941,31): text "Servis komunikace"; opens ServisNovaProdejna; tooltip Back to home page
rectangle at (960,70)-(1131,91): alarm colour if OUTVnitrniSvetla1; taps INVnitrniSvetla1; tooltip Kliknutím zapínáte a vypínáte svìtla DALI
rectangle at (810,70)-(951,91): text "Vnitrni svetla 1"
rectangle at (810,100)-(951,121): text "Vnitrni svetla 2"
rectangle at (810,130)-(951,151): text "Vnitrni svetla 3"
rectangle at (810,160)-(1121,181): text "Vnitrni reklama nad okny nocni osvìtleni"
rectangle at (820,190)-(961,211): text "Venkovni reklama 1"
rectangle at (820,220)-(961,241): text "Venkovni reklama 2"
rectangle at (820,250)-(961,271): text "Venkovni reklama 3"
rectangle at (820,280)-(961,301): text "Topeni okap 1"
rectangle at (820,310)-(961,331): text "Topeni okap 2"
rectangle at (820,340)-(981,361): text "Zásuvky 1 denni provoz"
rectangle at (820,370)-(961,391): text "Nouzove osvetleni"
rectangle at (820,400)-(1021,421): text "Vnitrni zasuvky denni provoz"
rectangle at (830,430)-(971,451): text "Venkobni reklama"
rectangle at (830,460)-(971,481): text "Topeni okap"
rectangle at (960,100)-(1131,121): alarm colour if OUTVnitrniSvetla2; taps INVnitrniSvetla2; tooltip Kliknutím zapínáte a vypínáte svìtla DALI
rectangle at (960,130)-(1131,151): alarm colour if OUTVnitrniSvetla3; taps INVnitrniSvetla3; tooltip Kliknutím zapínáte a vypínáte svìtla DALI
rectangle at (1110,160)-(1281,181): alarm colour if OUTVnitrniReklama; taps INVnitrniReklama; tooltip Kliknutím zapínáte a vypínáte svìtla DALI
rectangle at (960,190)-(1131,211): alarm colour if OUTVenkovniReklama1; taps INVenkovniReklama; tooltip Kliknutím zapínáte a vypínáte svìtla DALI
rectangle at (960,220)-(1131,241): alarm colour if OUTVenkovniReklama2; taps INVenkovniReklama; tooltip Kliknutím zapínáte a vypínáte svìtla DALI
rectangle at (960,250)-(1131,271): alarm colour if OUTVenkovniReklama3; taps INVenkovniReklama; tooltip Kliknutím zapínáte a vypínáte svìtla DALI
rectangle at (960,280)-(1131,301): alarm colour if OUTTopeniOkap1; taps INTopeniOkap; tooltip Kliknutím zapínáte a vypínáte svìtla DALI
rectangle at (960,310)-(1131,331): alarm colour if OUTTopeniOkap2; taps INTopeniOkap; tooltip Kliknutím zapínáte a vypínáte svìtla DALI
rectangle at (960,460)-(1131,481): alarm colour if OUTTopeniOkap; taps INTopeniOkap; tooltip Kliknutím zapínáte a vypínáte svìtla DALI
rectangle at (990,340)-(1161,361): alarm colour if OUTZasuvky1; tooltip Kliknutím zapínáte a vypínáte svìtla DALI
rectangle at (960,370)-(1131,391): alarm colour if OUTNouzoveOsvetleni; tooltip Kliknutím zapínáte a vypínáte svìtla DALI
rectangle at (1020,400)-(1191,421): alarm colour if OUTVnitrniZasuvkyDenniProvoz; taps INVnitrniZasuvkyDenniProvoz; tooltip Kliknutím zapínáte a vypínáte svìtla DALI
rectangle at (970,430)-(1141,451): alarm colour if OUTVnitrniReklama; taps INVnitrniReklama; tooltip Kliknutím zapínáte a vypínáte svìtla DALI
rectangle at (50,400)-(131,421): text "Nastaveni"; opens prodej_materialu_nastaveni; tooltip Back to home page
10 more shapes without text or variables
*)

(* Visualisation prodej_materialu_nastaveni
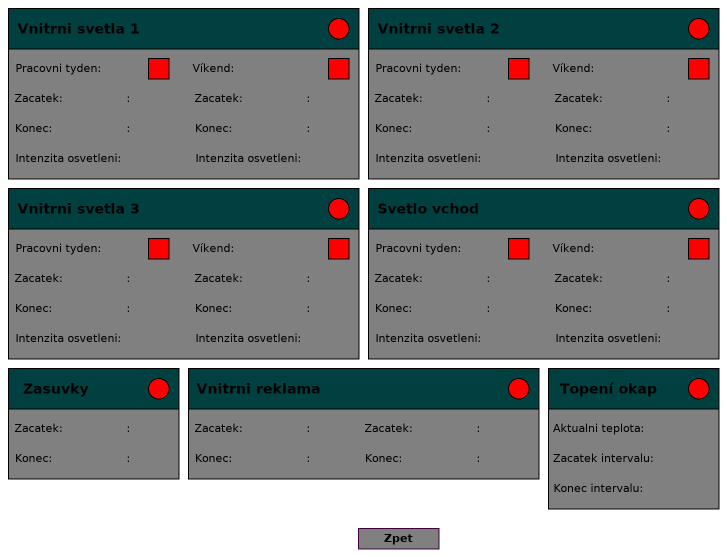
rectangle at (10,10)-(151,51): text "Vnitrni svetla 1"
ellipse at (330,20)-(351,41): alarm colour if ProdejnaMaterialu.PRGVnitrniSvetla1; toggles ProdejnaMaterialu.PRGVnitrniSvetla1
rectangle at (10,90)-(71,111): text "Zacatek:"
rectangle at (10,120)-(61,141): text "Konec:"
rectangle at (120,90)-(141,111): text ":"
rectangle at (120,120)-(141,141): text ":"
rectangle at (10,370)-(111,411): text "Zasuvky"
ellipse at (150,380)-(171,401): alarm colour if ProdejnaMaterialu.PRGVnitrniZasuvkyDenniProvoz; toggles ProdejnaMaterialu.PRGVnitrniZasuvkyDenniProvoz
rectangle at (10,420)-(71,441): text "Zacatek:"
rectangle at (10,450)-(61,471): text "Konec:"
rectangle at (120,420)-(141,441): text ":"
rectangle at (120,450)-(141,471): text ":"
rectangle at (370,190)-(491,231): text "Svetlo vchod"
ellipse at (690,200)-(711,221): alarm colour if ProdejnaMaterialu.PRGSvetloNadVchodem; toggles ProdejnaMaterialu.PRGSvetloNadVchodem
rectangle at (370,270)-(431,291): text "Zacatek:"
rectangle at (370,300)-(421,321): text "Konec:"
rectangle at (480,270)-(501,291): text ":"
rectangle at (480,300)-(501,321): text ":"
rectangle at (190,370)-(331,411): text "Vnitrni reklama"
ellipse at (510,380)-(531,401): alarm colour if ProdejnaMaterialu.PRGVnitrniReklama; toggles ProdejnaMaterialu.PRGVnitrniReklama
rectangle at (190,420)-(251,441): text "Zacatek:"
rectangle at (190,450)-(241,471): text "Konec:"
rectangle at (300,420)-(321,441): text ":"
rectangle at (300,450)-(321,471): text ":"
rectangle at (360,420)-(421,441): text "Zacatek:"
rectangle at (360,450)-(411,471): text "Konec:"
rectangle at (470,420)-(491,441): text ":"
rectangle at (470,450)-(491,471): text ":"
rectangle at (550,370)-(671,411): text "Topení okap"
ellipse at (690,380)-(711,401): alarm colour if INTopeniOkap
rectangle at (550,420)-(651,441): text "Aktualni teplota:"
rectangle at (550,450)-(661,471): text "Zacatek intervalu:"; tooltip Nejnižší teplota.
rectangle at (550,480)-(651,501): text "Konec intervalu:"; tooltip Nevyšší teplota.
rectangle at (10,150)-(131,171): text "Intenzita osvetleni:"
rectangle at (370,330)-(491,351): text "Intenzita osvetleni:"
rectangle at (370,240)-(471,261): text "Pracovni tyden:"
rectangle at (510,240)-(531,261): alarm colour if ProdejnaMaterialu.xSvetloNadVchodemPracTyden; toggles ProdejnaMaterialu.xSvetloNadVchodemPracTyden
rectangle at (550,270)-(611,291): text "Zacatek:"
rectangle at (550,300)-(601,321): text "Konec:"
rectangle at (660,270)-(681,291): text ":"
rectangle at (660,300)-(681,321): text ":"
rectangle at (550,330)-(671,351): text "Intenzita osvetleni:"
rectangle at (550,240)-(601,261): text "Víkend:"
rectangle at (690,240)-(711,261): alarm colour if ProdejnaMaterialu.xSvetloNadVchodemVikend; toggles ProdejnaMaterialu.xSvetloNadVchodemVikend
rectangle at (10,60)-(111,81): text "Pracovni tyden:"
rectangle at (150,60)-(171,81): alarm colour if ProdejnaMaterialu.xVnitrniSvetla1PracDen; toggles ProdejnaMaterialu.xVnitrniSvetla1PracDen
rectangle at (190,60)-(241,81): text "Víkend:"
rectangle at (330,60)-(351,81): alarm colour if ProdejnaMaterialu.xVnitrniSvetla1Vikend; toggles ProdejnaMaterialu.xVnitrniSvetla1Vikend
rectangle at (190,90)-(251,111): text "Zacatek:"
rectangle at (190,120)-(241,141): text "Konec:"
rectangle at (300,90)-(321,111): text ":"
rectangle at (300,120)-(321,141): text ":"
rectangle at (190,150)-(311,171): text "Intenzita osvetleni:"
rectangle at (370,10)-(511,51): text "Vnitrni svetla 2"
ellipse at (690,20)-(711,41): alarm colour if ProdejnaMaterialu.PRGVnitrniSvetla2; toggles ProdejnaMaterialu.PRGVnitrniSvetla2
rectangle at (370,90)-(431,111): text "Zacatek:"
rectangle at (370,120)-(421,141): text "Konec:"
rectangle at (480,90)-(501,111): text ":"
rectangle at (480,120)-(501,141): text ":"
rectangle at (370,150)-(491,171): text "Intenzita osvetleni:"
rectangle at (370,60)-(471,81): text "Pracovni tyden:"
rectangle at (510,60)-(531,81): alarm colour if ProdejnaMaterialu.xVnitrniSvetla2PracDen; toggles ProdejnaMaterialu.xVnitrniSvetla2PracDen
rectangle at (550,60)-(601,81): text "Víkend:"
rectangle at (690,60)-(711,81): alarm colour if ProdejnaMaterialu.xVnitrniSvetla2Vikend; toggles ProdejnaMaterialu.xVnitrniSvetla2Vikend
rectangle at (550,90)-(611,111): text "Zacatek:"
rectangle at (550,120)-(601,141): text "Konec:"
rectangle at (660,90)-(681,111): text ":"
rectangle at (660,120)-(681,141): text ":"
rectangle at (550,150)-(671,171): text "Intenzita osvetleni:"
rectangle at (10,190)-(151,231): text "Vnitrni svetla 3"
ellipse at (330,200)-(351,221): alarm colour if ProdejnaMaterialu.PRGVnitrniSvetla3; toggles ProdejnaMaterialu.PRGVnitrniSvetla3
rectangle at (10,270)-(71,291): text "Zacatek:"
rectangle at (10,300)-(61,321): text "Konec:"
rectangle at (120,270)-(141,291): text ":"
rectangle at (120,300)-(141,321): text ":"
rectangle at (10,330)-(131,351): text "Intenzita osvetleni:"
rectangle at (10,240)-(111,261): text "Pracovni tyden:"
rectangle at (150,240)-(171,261): alarm colour if ProdejnaMaterialu.xVnitrniSvetla3PracDen; toggles ProdejnaMaterialu.xVnitrniSvetla3PracDen
rectangle at (190,240)-(241,261): text "Víkend:"
rectangle at (330,240)-(351,261): alarm colour if ProdejnaMaterialu.xVnitrniSvetla3Vikend; toggles ProdejnaMaterialu.xVnitrniSvetla3Vikend
rectangle at (190,270)-(251,291): text "Zacatek:"
rectangle at (190,300)-(241,321): text "Konec:"
rectangle at (300,270)-(321,291): text ":"
rectangle at (300,300)-(321,321): text ":"
rectangle at (190,330)-(311,351): text "Intenzita osvetleni:"
rectangle at (360,530)-(441,551): text "Zpet"; opens prodej_materialu; tooltip Back to home page
14 more shapes without text or variables
55 elements of other kinds (tables, trends, ...) not read
*)

(* Visualisation prodej_svetel
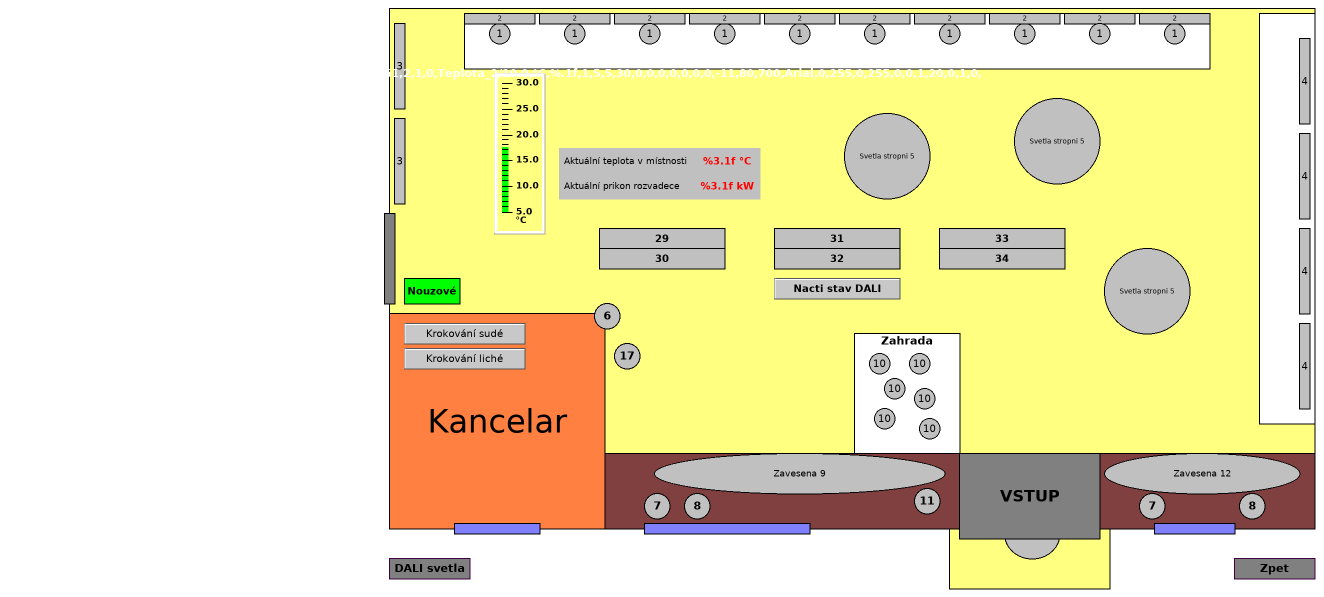
rounded rectangle at (485,345)-(591,476): text "Zahrada"
ellipse at (635,520)-(691,571): alarm colour if .KA13; taps .TL10s; tooltip Dlouhý stisk zapne svìtlo. (cca 1s)
rectangle at (25,130)-(36,216): text "3"; alarm colour if .KA03
rectangle at (35,290)-(91,316): text "Nouzové"; alarm colour if .KA20
rectangle at (20,325)-(236,541): text "Kancelar"
rectangle at (865,570)-(946,591): text "Zpet"; opens PLC_VISU; tooltip Back to home page
ellipse at (315,505)-(341,531): text "8"; alarm colour if .ka08
ellipse at (735,465)-(931,506): text "Zavesena 12"; alarm colour if .KA12
rectangle at (930,50)-(941,136): text "4"; alarm colour if .KA04
ellipse at (500,365)-(521,386): text "10"; alarm colour if .KA10
ellipse at (285,465)-(576,506): text "Zavesena 9"; alarm colour if .KA09
rectangle at (590,465)-(731,551): text "VSTUP"
rectangle at (325,160)-(391,186): text "%3.1f °C"; shows .Teplota_2/10.0
rectangle at (190,160)-(326,186): text "Aktuální teplota v místnosti"
ellipse at (120,35)-(141,56): text "1"; alarm colour if .KA01; taps .TL10s; tooltip Klinutím zapínáte žárovky na deskách
rectangle at (95,25)-(166,36): text "2"; alarm colour if .KA02
ellipse at (275,505)-(301,531): text "7"; alarm colour if .ka07
ellipse at (870,505)-(896,531): text "8"; alarm colour if .ka08
ellipse at (770,505)-(796,531): text "7"; alarm colour if .ka07
rectangle at (930,145)-(941,231): text "4"; alarm colour if .KA04
rectangle at (930,335)-(941,421): text "4"; alarm colour if .KA04
rectangle at (930,240)-(941,326): text "4"; alarm colour if .KA04
rectangle at (25,35)-(36,121): text "3"; alarm colour if .KA03
rectangle at (190,185)-(326,211): text "Aktuální prikon rozvadece"
rectangle at (325,185)-(391,211): text "%3.1f kW"; shows TriFaze.arVykon[1]+TriFaze.arVykon[2]+TriFaze.arVykon[3]
button at (35,335)-(156,356): text "Krokování sudé"; taps .TL08s; tooltip Kliknutím krokujete sudé releové výstupy oovládající svìtla.
button at (35,360)-(156,381): text "Krokování liché"; taps .TL07s; tooltip Kliknutím krokujete liché releové výstupy oovládající svìtla.
rectangle at (230,240)-(356,261): text "29"; alarm colour if DALI_Config.Kurzadr[29]
rectangle at (230,240)-(356,261): text "29"; invisible if not DALI_Config.Kurzadr[29]; alarm colour if DALI_Config.LampeEin[29]; taps .TL09s; tooltip Kliknutím zapínáte a vypínáte svìtla DALI
rectangle at (230,260)-(356,281): text "30"; alarm colour if DALI_Config.Kurzadr[30]
rectangle at (230,260)-(356,281): text "30"; invisible if not DALI_Config.Kurzadr[30]; alarm colour if DALI_Config.LampeEin[30]; taps .TL09s; tooltip Kliknutím zapínáte a vypínáte svìtla DALI
rectangle at (405,240)-(531,261): text "31"; alarm colour if DALI_Config.Kurzadr[31]
rectangle at (405,240)-(531,261): text "31"; invisible if not DALI_Config.Kurzadr[31]; alarm colour if DALI_Config.LampeEin[31]; taps .TL09s; tooltip Kliknutím zapínáte a vypínáte svìtla DALI
rectangle at (405,260)-(531,281): text "32"; alarm colour if DALI_Config.Kurzadr[32]
rectangle at (405,260)-(531,281): text "32"; invisible if not DALI_Config.Kurzadr[32]; alarm colour if DALI_Config.LampeEin[32]; taps .TL09s; tooltip Kliknutím zapínáte a vypínáte svìtla DALI
rectangle at (570,240)-(696,261): text "33"; alarm colour if DALI_Config.Kurzadr[33]
rectangle at (570,240)-(696,261): text "33"; invisible if not DALI_Config.Kurzadr[33]; alarm colour if DALI_Config.LampeEin[33]; taps .TL09s; tooltip Kliknutím zapínáte a vypínáte svìtla DALI
rectangle at (570,260)-(696,281): text "34"; alarm colour if DALI_Config.Kurzadr[34]
rectangle at (570,260)-(696,281): text "34"; invisible if not DALI_Config.Kurzadr[34]; alarm colour if DALI_Config.LampeEin[34]; taps .TL09s; tooltip Kliknutím zapínáte a vypínáte svìtla DALI
button at (405,290)-(531,311): text "Nacti stav DALI"; taps DALI_Config.Status; tooltip Kliknutim nactete status svetel. (sviti, nesviti, vadna).
rectangle at (245,25)-(316,36): text "2"; alarm colour if .KA02
ellipse at (195,35)-(216,56): text "1"; alarm colour if .KA01; taps .TL10s; tooltip Klinutím zapínáte žárovky na deskách
rectangle at (170,25)-(241,36): text "2"; alarm colour if .KA02
ellipse at (270,35)-(291,56): text "1"; alarm colour if .KA01; taps .TL10s; tooltip Klinutím zapínáte žárovky na deskách
ellipse at (345,35)-(366,56): text "1"; alarm colour if .KA01; taps .TL10s; tooltip Klinutím zapínáte žárovky na deskách
rectangle at (320,25)-(391,36): text "2"; alarm colour if .KA02
rectangle at (470,25)-(541,36): text "2"; alarm colour if .KA02
ellipse at (420,35)-(441,56): text "1"; alarm colour if .KA01; taps .TL10s; tooltip Klinutím zapínáte žárovky na deskách
rectangle at (395,25)-(466,36): text "2"; alarm colour if .KA02
ellipse at (495,35)-(516,56): text "1"; alarm colour if .KA01; taps .TL10s; tooltip Klinutím zapínáte žárovky na deskách
ellipse at (570,35)-(591,56): text "1"; alarm colour if .KA01; taps .TL10s; tooltip Klinutím zapínáte žárovky na deskách
rectangle at (545,25)-(616,36): text "2"; alarm colour if .KA02
rectangle at (695,25)-(766,36): text "2"; alarm colour if .KA02
ellipse at (645,35)-(666,56): text "1"; alarm colour if .KA01; taps .TL10s; tooltip Klinutím zapínáte žárovky na deskách
rectangle at (620,25)-(691,36): text "2"; alarm colour if .KA02
ellipse at (720,35)-(741,56): text "1"; alarm colour if .KA01; taps .TL10s; tooltip Klinutím zapínáte žárovky na deskách
ellipse at (795,35)-(816,56): text "1"; alarm colour if .KA01; taps .TL10s; tooltip Klinutím zapínáte žárovky na deskách
rectangle at (770,25)-(841,36): text "2"; alarm colour if .KA02
ellipse at (475,125)-(561,211): text "Svetla stropni 5"; alarm colour if .KA05
ellipse at (645,110)-(731,196): text "Svetla stropni 5"; alarm colour if .KA05
ellipse at (735,260)-(821,346): text "Svetla stropni 5"; alarm colour if .KA05
ellipse at (505,420)-(526,441): text "10"; alarm colour if .KA10
ellipse at (545,400)-(566,421): text "10"; alarm colour if .KA10
ellipse at (540,365)-(561,386): text "10"; alarm colour if .KA10
ellipse at (550,430)-(571,451): text "10"; alarm colour if .KA10
ellipse at (515,390)-(536,411): text "10"; alarm colour if .KA10
ellipse at (225,315)-(251,341): text "6"; alarm colour if .ka06
ellipse at (545,500)-(571,526): text "11"; alarm colour if .ka11
ellipse at (245,355)-(271,381): text "17"; alarm colour if .ka17
group at (125,85)-(176,246)
  rectangle at (0,0)-(1,1): text "{ExtendedElement},Visu\ElementDLL.ete,1,@Bargraph,51,161,2,1,0,Teplota_2/10.0,°C,%.1f,1,5,5,30,0,0,0,0,0,0,0,-11,80,700,Arial,0,255,0,255,0,0,1,20,0,1,0,"
  rectangle at (8,74)-(14,139): alarm colour if (Teplota_2/10.0) > 20; top ((Teplota_2/10.0 * 1.0) - 17.5)  * -5.2
  rectangle at (20,129)-(47,148): text "5.0"
  rectangle at (20,103)-(47,122): text "10.0"
  rectangle at (20,77)-(47,96): text "15.0"
  rectangle at (20,52)-(47,71): text "20.0"
  rectangle at (20,26)-(47,45): text "25.0"
  rectangle at (20,0)-(47,19): text "30.0"
  rectangle at (15,140)-(39,154): text "°C"
rectangle at (20,570)-(101,591): text "DALI svetla"; opens DALI_cfg; tooltip Back to home page
44 more shapes without text or variables
*)

(* Visualisation Scene_configuration
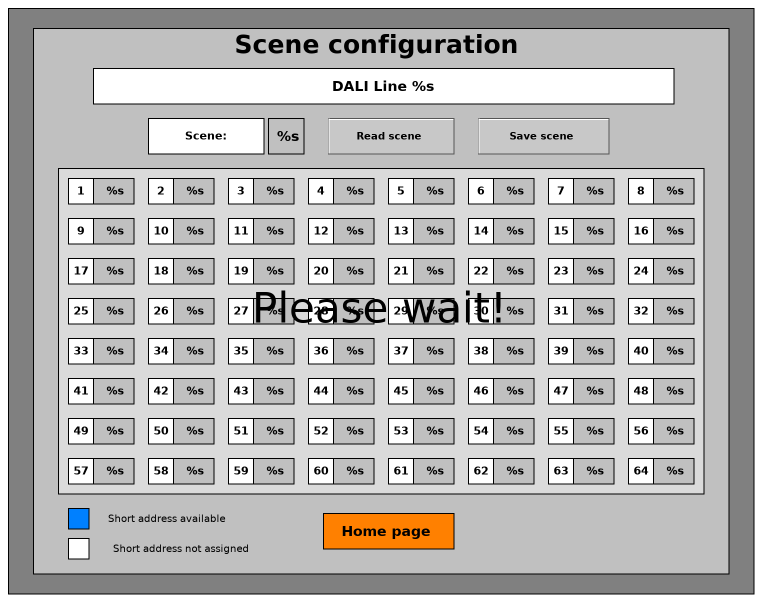
rectangle at (50,25)-(746,571): text "Scene configuration"
rounded rectangle at (340,510)-(471,546): text "Home page"; opens DALI; tooltip Back to home page
rounded rectangle at (110,65)-(691,101): text "DALI Line %s"; shows DALI_Config.bDali_Linie; tooltip You can change the DALI Line only on the home page.
rectangle at (85,175)-(111,201): text "1"; alarm colour if Dali_Config.Kurzadr[1]
rectangle at (110,175)-(151,201): text "%s"; shows DALI_Config.Szenenwert[1]; tooltip 0 % = Off 1 - 100 % = Dim level 101 % = Mask; editable
button at (495,115)-(626,151): text "Save scene"; taps DALI_Config.SzeneSpeichern; tooltip Save the configured dim levels in the ECGs.
button at (345,115)-(471,151): text "Read scene"; taps DALI_Config.SzeneLesen; tooltip Read the saved scene values from the ECGs.
rectangle at (85,215)-(111,241): text "9"; alarm colour if Dali_Config.Kurzadr[9]
rectangle at (110,215)-(151,241): text "%s"; shows DALI_Config.Szenenwert[9]; tooltip 0 % = Off 1 - 100 % = Dim level 101 % = Mask; editable
rectangle at (85,255)-(111,281): text "17"; alarm colour if Dali_Config.Kurzadr[17]
rectangle at (110,255)-(151,281): text "%s"; shows DALI_Config.Szenenwert[17]; tooltip 0 % = Off 1 - 100 % = Dim level 101 % = Mask; editable
rectangle at (85,295)-(111,321): text "25"; alarm colour if Dali_Config.Kurzadr[25]
rectangle at (110,295)-(151,321): text "%s"; shows DALI_Config.Szenenwert[25]; tooltip 0 % = Off 1 - 100 % = Dim level 101 % = Mask; editable
rectangle at (85,335)-(111,361): text "33"; alarm colour if Dali_Config.Kurzadr[33]
rectangle at (110,335)-(151,361): text "%s"; shows DALI_Config.Szenenwert[33]; tooltip 0 % = Off 1 - 100 % = Dim level 101 % = Mask; editable
rectangle at (85,375)-(111,401): text "41"; alarm colour if Dali_Config.Kurzadr[41]
rectangle at (110,375)-(151,401): text "%s"; shows DALI_Config.Szenenwert[41]; tooltip 0 % = Off 1 - 100 % = Dim level 101 % = Mask; editable
rectangle at (85,415)-(111,441): text "49"; alarm colour if Dali_Config.Kurzadr[49]
rectangle at (110,415)-(151,441): text "%s"; shows DALI_Config.Szenenwert[49]; tooltip 0 % = Off 1 - 100 % = Dim level 101 % = Mask; editable
rectangle at (85,455)-(111,481): text "57"; alarm colour if Dali_Config.Kurzadr[57]
rectangle at (110,455)-(151,481): text "%s"; shows DALI_Config.Szenenwert[57]; tooltip 0 % = Off 1 - 100 % = Dim level 101 % = Mask; editable
rectangle at (165,175)-(191,201): text "2"; alarm colour if Dali_Config.Kurzadr[2]
rectangle at (190,175)-(231,201): text "%s"; shows DALI_Config.Szenenwert[2]; tooltip 0 % = Off 1 - 100 % = Dim level 101 % = Mask; editable
rectangle at (165,215)-(191,241): text "10"; alarm colour if Dali_Config.Kurzadr[10]
rectangle at (190,215)-(231,241): text "%s"; shows DALI_Config.Szenenwert[10]; tooltip 0 % = Off 1 - 100 % = Dim level 101 % = Mask; editable
rectangle at (165,255)-(191,281): text "18"; alarm colour if Dali_Config.Kurzadr[18]
rectangle at (190,255)-(231,281): text "%s"; shows DALI_Config.Szenenwert[18]; tooltip 0 % = Off 1 - 100 % = Dim level 101 % = Mask; editable
rectangle at (165,295)-(191,321): text "26"; alarm colour if Dali_Config.Kurzadr[26]
rectangle at (190,295)-(231,321): text "%s"; shows DALI_Config.Szenenwert[26]; tooltip 0 % = Off 1 - 100 % = Dim level 101 % = Mask; editable
rectangle at (165,335)-(191,361): text "34"; alarm colour if Dali_Config.Kurzadr[34]
rectangle at (190,335)-(231,361): text "%s"; shows DALI_Config.Szenenwert[34]; tooltip 0 % = Off 1 - 100 % = Dim level 101 % = Mask; editable
rectangle at (165,375)-(191,401): text "42"; alarm colour if Dali_Config.Kurzadr[42]
rectangle at (190,375)-(231,401): text "%s"; shows DALI_Config.Szenenwert[42]; tooltip 0 % = Off 1 - 100 % = Dim level 101 % = Mask; editable
rectangle at (165,415)-(191,441): text "50"; alarm colour if Dali_Config.Kurzadr[50]
rectangle at (190,415)-(231,441): text "%s"; shows DALI_Config.Szenenwert[50]; tooltip 0 % = Off 1 - 100 % = Dim level 101 % = Mask; editable
rectangle at (165,455)-(191,481): text "58"; alarm colour if Dali_Config.Kurzadr[58]
rectangle at (190,455)-(231,481): text "%s"; shows DALI_Config.Szenenwert[58]; tooltip 0 % = Off 1 - 100 % = Dim level 101 % = Mask; editable
rectangle at (245,175)-(271,201): text "3"; alarm colour if Dali_Config.Kurzadr[3]
rectangle at (270,175)-(311,201): text "%s"; shows DALI_Config.Szenenwert[3]; tooltip 0 % = Off 1 - 100 % = Dim level 101 % = Mask; editable
rectangle at (245,215)-(271,241): text "11"; alarm colour if Dali_Config.Kurzadr[11]
rectangle at (270,215)-(311,241): text "%s"; shows DALI_Config.Szenenwert[11]; tooltip 0 % = Off 1 - 100 % = Dim level 101 % = Mask; editable
rectangle at (245,255)-(271,281): text "19"; alarm colour if Dali_Config.Kurzadr[19]
rectangle at (270,255)-(311,281): text "%s"; shows DALI_Config.Szenenwert[19]; tooltip 0 % = Off 1 - 100 % = Dim level 101 % = Mask; editable
rectangle at (245,295)-(271,321): text "27"; alarm colour if Dali_Config.Kurzadr[27]
rectangle at (270,295)-(311,321): text "%s"; shows DALI_Config.Szenenwert[27]; tooltip 0 % = Off 1 - 100 % = Dim level 101 % = Mask; editable
rectangle at (245,335)-(271,361): text "35"; alarm colour if Dali_Config.Kurzadr[35]
rectangle at (270,335)-(311,361): text "%s"; shows DALI_Config.Szenenwert[35]; tooltip 0 % = Off 1 - 100 % = Dim level 101 % = Mask; editable
rectangle at (245,375)-(271,401): text "43"; alarm colour if Dali_Config.Kurzadr[43]
rectangle at (270,375)-(311,401): text "%s"; shows DALI_Config.Szenenwert[43]; tooltip 0 % = Off 1 - 100 % = Dim level 101 % = Mask; editable
rectangle at (245,415)-(271,441): text "51"; alarm colour if Dali_Config.Kurzadr[51]
rectangle at (270,415)-(311,441): text "%s"; shows DALI_Config.Szenenwert[51]; tooltip 0 % = Off 1 - 100 % = Dim level 101 % = Mask; editable
rectangle at (245,455)-(271,481): text "59"; alarm colour if Dali_Config.Kurzadr[59]
rectangle at (270,455)-(311,481): text "%s"; shows DALI_Config.Szenenwert[59]; tooltip 0 % = Off 1 - 100 % = Dim level 101 % = Mask; editable
rectangle at (325,175)-(351,201): text "4"; alarm colour if Dali_Config.Kurzadr[4]
rectangle at (350,175)-(391,201): text "%s"; shows DALI_Config.Szenenwert[4]; tooltip 0 % = Off 1 - 100 % = Dim level 101 % = Mask; editable
rectangle at (325,215)-(351,241): text "12"; alarm colour if Dali_Config.Kurzadr[12]
rectangle at (350,215)-(391,241): text "%s"; shows DALI_Config.Szenenwert[12]; tooltip 0 % = Off 1 - 100 % = Dim level 101 % = Mask; editable
rectangle at (325,255)-(351,281): text "20"; alarm colour if Dali_Config.Kurzadr[20]
rectangle at (350,255)-(391,281): text "%s"; shows DALI_Config.Szenenwert[20]; tooltip 0 % = Off 1 - 100 % = Dim level 101 % = Mask; editable
rectangle at (325,295)-(351,321): text "28"; alarm colour if Dali_Config.Kurzadr[28]
rectangle at (350,295)-(391,321): text "%s"; shows DALI_Config.Szenenwert[28]; tooltip 0 % = Off 1 - 100 % = Dim level 101 % = Mask; editable
rectangle at (325,335)-(351,361): text "36"; alarm colour if Dali_Config.Kurzadr[36]
rectangle at (350,335)-(391,361): text "%s"; shows DALI_Config.Szenenwert[36]; tooltip 0 % = Off 1 - 100 % = Dim level 101 % = Mask; editable
rectangle at (325,375)-(351,401): text "44"; alarm colour if Dali_Config.Kurzadr[44]
rectangle at (350,375)-(391,401): text "%s"; shows DALI_Config.Szenenwert[44]; tooltip 0 % = Off 1 - 100 % = Dim level 101 % = Mask; editable
rectangle at (325,415)-(351,441): text "52"; alarm colour if Dali_Config.Kurzadr[52]
rectangle at (350,415)-(391,441): text "%s"; shows DALI_Config.Szenenwert[52]; tooltip 0 % = Off 1 - 100 % = Dim level 101 % = Mask; editable
rectangle at (325,455)-(351,481): text "60"; alarm colour if Dali_Config.Kurzadr[60]
rectangle at (350,455)-(391,481): text "%s"; shows DALI_Config.Szenenwert[60]; tooltip 0 % = Off 1 - 100 % = Dim level 101 % = Mask; editable
rectangle at (405,175)-(431,201): text "5"; alarm colour if Dali_Config.Kurzadr[5]
rectangle at (430,175)-(471,201): text "%s"; shows DALI_Config.Szenenwert[5]; tooltip 0 % = Off 1 - 100 % = Dim level 101 % = Mask; editable
rectangle at (405,215)-(431,241): text "13"; alarm colour if Dali_Config.Kurzadr[13]
rectangle at (430,215)-(471,241): text "%s"; shows DALI_Config.Szenenwert[13]; tooltip 0 % = Off 1 - 100 % = Dim level 101 % = Mask; editable
rectangle at (405,255)-(431,281): text "21"; alarm colour if Dali_Config.Kurzadr[21]
rectangle at (430,255)-(471,281): text "%s"; shows DALI_Config.Szenenwert[21]; tooltip 0 % = Off 1 - 100 % = Dim level 101 % = Mask; editable
rectangle at (405,295)-(431,321): text "29"; alarm colour if Dali_Config.Kurzadr[29]
rectangle at (430,295)-(471,321): text "%s"; shows DALI_Config.Szenenwert[29]; tooltip 0 % = Off 1 - 100 % = Dim level 101 % = Mask; editable
rectangle at (405,335)-(431,361): text "37"; alarm colour if Dali_Config.Kurzadr[37]
rectangle at (430,335)-(471,361): text "%s"; shows DALI_Config.Szenenwert[37]; tooltip 0 % = Off 1 - 100 % = Dim level 101 % = Mask; editable
rectangle at (405,375)-(431,401): text "45"; alarm colour if Dali_Config.Kurzadr[45]
rectangle at (430,375)-(471,401): text "%s"; shows DALI_Config.Szenenwert[45]; tooltip 0 % = Off 1 - 100 % = Dim level 101 % = Mask; editable
rectangle at (405,415)-(431,441): text "53"; alarm colour if Dali_Config.Kurzadr[53]
rectangle at (430,415)-(471,441): text "%s"; shows DALI_Config.Szenenwert[53]; tooltip 0 % = Off 1 - 100 % = Dim level 101 % = Mask; editable
rectangle at (405,455)-(431,481): text "61"; alarm colour if Dali_Config.Kurzadr[61]
rectangle at (430,455)-(471,481): text "%s"; shows DALI_Config.Szenenwert[61]; tooltip 0 % = Off 1 - 100 % = Dim level 101 % = Mask; editable
rectangle at (485,175)-(511,201): text "6"; alarm colour if Dali_Config.Kurzadr[6]
rectangle at (510,175)-(551,201): text "%s"; shows DALI_Config.Szenenwert[6]; tooltip 0 % = Off 1 - 100 % = Dim level 101 % = Mask; editable
rectangle at (485,215)-(511,241): text "14"; alarm colour if Dali_Config.Kurzadr[14]
rectangle at (510,215)-(551,241): text "%s"; shows DALI_Config.Szenenwert[14]; tooltip 0 % = Off 1 - 100 % = Dim level 101 % = Mask; editable
rectangle at (485,255)-(511,281): text "22"; alarm colour if Dali_Config.Kurzadr[22]
rectangle at (510,255)-(551,281): text "%s"; shows DALI_Config.Szenenwert[22]; tooltip 0 % = Off 1 - 100 % = Dim level 101 % = Mask; editable
rectangle at (485,295)-(511,321): text "30"; alarm colour if Dali_Config.Kurzadr[30]
rectangle at (510,295)-(551,321): text "%s"; shows DALI_Config.Szenenwert[30]; tooltip 0 % = Off 1 - 100 % = Dim level 101 % = Mask; editable
rectangle at (485,335)-(511,361): text "38"; alarm colour if Dali_Config.Kurzadr[38]
rectangle at (510,335)-(551,361): text "%s"; shows DALI_Config.Szenenwert[38]; tooltip 0 % = Off 1 - 100 % = Dim level 101 % = Mask; editable
rectangle at (485,375)-(511,401): text "46"; alarm colour if Dali_Config.Kurzadr[46]
rectangle at (510,375)-(551,401): text "%s"; shows DALI_Config.Szenenwert[46]; tooltip 0 % = Off 1 - 100 % = Dim level 101 % = Mask; editable
rectangle at (485,415)-(511,441): text "54"; alarm colour if Dali_Config.Kurzadr[54]
rectangle at (510,415)-(551,441): text "%s"; shows DALI_Config.Szenenwert[54]; tooltip 0 % = Off 1 - 100 % = Dim level 101 % = Mask; editable
rectangle at (485,455)-(511,481): text "62"; alarm colour if Dali_Config.Kurzadr[62]
rectangle at (510,455)-(551,481): text "%s"; shows DALI_Config.Szenenwert[62]; tooltip 0 % = Off 1 - 100 % = Dim level 101 % = Mask; editable
rectangle at (565,175)-(591,201): text "7"; alarm colour if Dali_Config.Kurzadr[7]
rectangle at (590,175)-(631,201): text "%s"; shows DALI_Config.Szenenwert[7]; tooltip 0 % = Off 1 - 100 % = Dim level 101 % = Mask; editable
rectangle at (565,215)-(591,241): text "15"; alarm colour if Dali_Config.Kurzadr[15]
rectangle at (590,215)-(631,241): text "%s"; shows DALI_Config.Szenenwert[15]; tooltip 0 % = Off 1 - 100 % = Dim level 101 % = Mask; editable
rectangle at (565,255)-(591,281): text "23"; alarm colour if Dali_Config.Kurzadr[23]
rectangle at (590,255)-(631,281): text "%s"; shows DALI_Config.Szenenwert[23]; tooltip 0 % = Off 1 - 100 % = Dim level 101 % = Mask; editable
rectangle at (565,295)-(591,321): text "31"; alarm colour if Dali_Config.Kurzadr[31]
rectangle at (590,295)-(631,321): text "%s"; shows DALI_Config.Szenenwert[31]; tooltip 0 % = Off 1 - 100 % = Dim level 101 % = Mask; editable
rectangle at (565,335)-(591,361): text "39"; alarm colour if Dali_Config.Kurzadr[39]
rectangle at (590,335)-(631,361): text "%s"; shows DALI_Config.Szenenwert[39]; tooltip 0 % = Off 1 - 100 % = Dim level 101 % = Mask; editable
rectangle at (565,375)-(591,401): text "47"; alarm colour if Dali_Config.Kurzadr[47]
rectangle at (590,375)-(631,401): text "%s"; shows DALI_Config.Szenenwert[47]; tooltip 0 % = Off 1 - 100 % = Dim level 101 % = Mask; editable
rectangle at (565,415)-(591,441): text "55"; alarm colour if Dali_Config.Kurzadr[55]
rectangle at (590,415)-(631,441): text "%s"; shows DALI_Config.Szenenwert[55]; tooltip 0 % = Off 1 - 100 % = Dim level 101 % = Mask; editable
rectangle at (565,455)-(591,481): text "63"; alarm colour if Dali_Config.Kurzadr[63]
rectangle at (590,455)-(631,481): text "%s"; shows DALI_Config.Szenenwert[63]; tooltip 0 % = Off 1 - 100 % = Dim level 101 % = Mask; editable
rectangle at (645,175)-(671,201): text "8"; alarm colour if Dali_Config.Kurzadr[8]
rectangle at (670,175)-(711,201): text "%s"; shows DALI_Config.Szenenwert[8]; tooltip 0 % = Off 1 - 100 % = Dim level 101 % = Mask; editable
rectangle at (645,215)-(671,241): text "16"; alarm colour if Dali_Config.Kurzadr[16]
rectangle at (670,215)-(711,241): text "%s"; shows DALI_Config.Szenenwert[16]; tooltip 0 % = Off 1 - 100 % = Dim level 101 % = Mask; editable
rectangle at (645,255)-(671,281): text "24"; alarm colour if Dali_Config.Kurzadr[24]
rectangle at (670,255)-(711,281): text "%s"; shows DALI_Config.Szenenwert[24]; tooltip 0 % = Off 1 - 100 % = Dim level 101 % = Mask; editable
rectangle at (645,295)-(671,321): text "32"; alarm colour if Dali_Config.Kurzadr[32]
rectangle at (670,295)-(711,321): text "%s"; shows DALI_Config.Szenenwert[32]; tooltip 0 % = Off 1 - 100 % = Dim level 101 % = Mask; editable
rectangle at (645,335)-(671,361): text "40"; alarm colour if Dali_Config.Kurzadr[40]
rectangle at (670,335)-(711,361): text "%s"; shows DALI_Config.Szenenwert[40]; tooltip 0 % = Off 1 - 100 % = Dim level 101 % = Mask; editable
rectangle at (645,375)-(671,401): text "48"; alarm colour if Dali_Config.Kurzadr[48]
rectangle at (670,375)-(711,401): text "%s"; shows DALI_Config.Szenenwert[48]; tooltip 0 % = Off 1 - 100 % = Dim level 101 % = Mask; editable
rectangle at (645,415)-(671,441): text "56"; alarm colour if Dali_Config.Kurzadr[56]
rectangle at (670,415)-(711,441): text "%s"; shows DALI_Config.Szenenwert[56]; tooltip 0 % = Off 1 - 100 % = Dim level 101 % = Mask; editable
rectangle at (645,455)-(671,481): text "64"; alarm colour if Dali_Config.Kurzadr[64]
rectangle at (670,455)-(711,481): text "%s"; shows DALI_Config.Szenenwert[64]; tooltip 0 % = Off 1 - 100 % = Dim level 101 % = Mask; editable
rectangle at (165,115)-(281,151): text "Scene:"
rectangle at (285,115)-(321,151): text "%s"; shows DALI_Config.Szene; tooltip Select scene 1 - 16; editable
rectangle at (110,505)-(261,526): text "Short address available"
rectangle at (105,535)-(291,556): text "Short address not assigned"
rectangle at (51,111)-(742,498): text "Please wait!"; invisible if NOT DALI_Config.Unsichtbar
4 more shapes without text or variables
*)

(* Visualisation ServisNovaProdejna
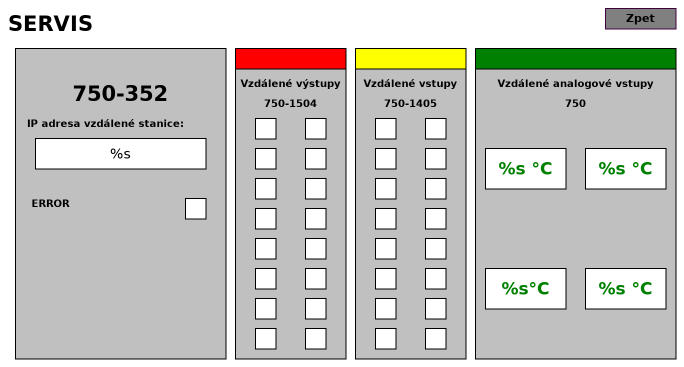
rectangle at (270,120)-(291,141): alarm colour if VzdalenyVystup1; toggles VzdalenyVystup1
rectangle at (250,70)-(361,101): text "Vzdálené výstupy"
rectangle at (320,120)-(341,141): alarm colour if VzdalenyVystup2; toggles VzdalenyVystup2
rectangle at (270,150)-(291,171): alarm colour if VzdalenyVystup3; toggles VzdalenyVystup3
rectangle at (320,150)-(341,171): alarm colour if VzdalenyVystup4; toggles VzdalenyVystup4
rectangle at (270,180)-(291,201): alarm colour if VzdalenyVystup5; toggles VzdalenyVystup5
rectangle at (320,180)-(341,201): alarm colour if VzdalenyVystup6; toggles VzdalenyVystup6
rectangle at (270,210)-(291,231): alarm colour if VzdalenyVystup7; toggles VzdalenyVystup7
rectangle at (320,210)-(341,231): alarm colour if VzdalenyVystup8; toggles VzdalenyVystup8
rectangle at (270,240)-(291,261): alarm colour if VzdalenyVystup9; toggles VzdalenyVystup9
rectangle at (320,240)-(341,261): alarm colour if VzdalenyVystup10; toggles VzdalenyVystup10
rectangle at (270,270)-(291,291): alarm colour if VzdalenyVystup11; toggles VzdalenyVystup11
rectangle at (320,270)-(341,291): alarm colour if VzdalenyVystup12; toggles VzdalenyVystup12
rectangle at (270,300)-(291,321): alarm colour if VzdalenyVystup13; toggles VzdalenyVystup13
rectangle at (320,300)-(341,321): alarm colour if VzdalenyVystup14; toggles VzdalenyVystup14
rectangle at (270,330)-(291,351): alarm colour if VzdalenyVystup15; toggles VzdalenyVystup15
rectangle at (320,330)-(341,351): alarm colour if VzdalenyVystup16; toggles VzdalenyVystup16
rectangle at (10,10)-(121,41): text "SERVIS"
rectangle at (250,90)-(361,121): text "750-1504"
rectangle at (390,120)-(411,141): alarm colour if VzdalenyVstup1
rectangle at (370,70)-(481,101): text "Vzdálené vstupy"
rectangle at (440,120)-(461,141): alarm colour if VzdalenyVstup2
rectangle at (390,150)-(411,171): alarm colour if VzdalenyVstup3
rectangle at (440,150)-(461,171): alarm colour if VzdalenyVstup4
rectangle at (390,180)-(411,201): alarm colour if VzdalenyVstup5
rectangle at (440,180)-(461,201): alarm colour if VzdalenyVstup6
rectangle at (390,210)-(411,231): alarm colour if VzdalenyVstup7
rectangle at (440,210)-(461,231): alarm colour if VzdalenyVstup8
rectangle at (390,240)-(411,261): alarm colour if VzdalenyVstup9
rectangle at (440,240)-(461,261): alarm colour if VzdalenyVstup10
rectangle at (390,270)-(411,291): alarm colour if VzdalenyVstup11
rectangle at (440,270)-(461,291): alarm colour if VzdalenyVstup12
rectangle at (390,300)-(411,321): alarm colour if VzdalenyVstup13
rectangle at (440,300)-(461,321): alarm colour if VzdalenyVstup14
rectangle at (390,330)-(411,351): alarm colour if VzdalenyVstup15
rectangle at (440,330)-(461,351): alarm colour if VzdalenyVstup16
rectangle at (370,90)-(481,121): text "750-1405"
rectangle at (30,80)-(241,111): text "750-352"
rectangle at (490,70)-(691,101): text "Vzdálené analogové vstupy"
rectangle at (490,90)-(691,121): text "750"
rectangle at (30,110)-(211,141): text "IP adresa vzdálené stanice:"
rectangle at (50,140)-(221,171): text "%s"; shows IPSlaveProdejnaMaterial
rounded rectangle at (500,150)-(581,191): text "%s °C"; shows VzdalenaTeplota1/10.0
rounded rectangle at (600,150)-(681,191): text "%s °C"; shows VzdalenaTeplota2/10.0
rounded rectangle at (500,270)-(581,311): text "%s°C"; shows VzdalenaTeplota3/10.0
rounded rectangle at (600,270)-(681,311): text "%s °C"; shows VzdalenaTeplota4/10.0
rectangle at (200,200)-(221,221): alarm colour if PLC_PRG.NoError
rectangle at (10,190)-(121,221): text "ERROR"
rectangle at (620,10)-(691,31): text "Zpet"; opens prodej_materialu; tooltip Back to home page
7 more shapes without text or variables
*)

(* Visualisation Sort_short_address
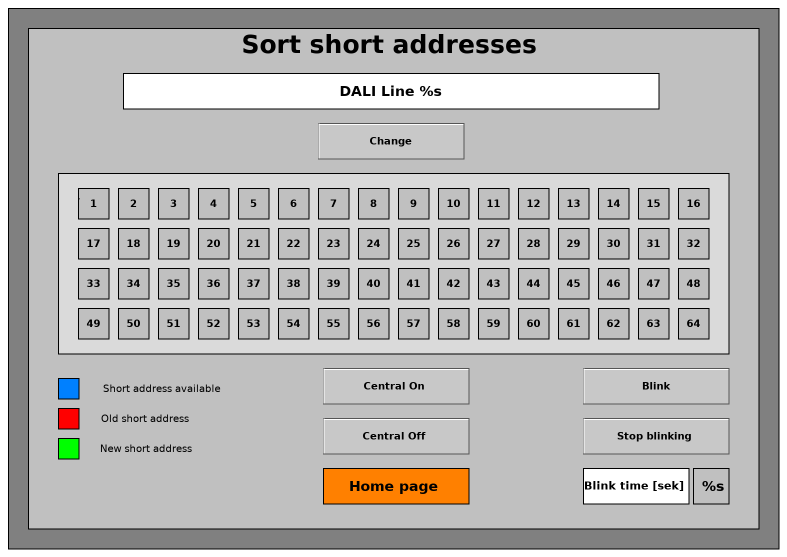
rectangle at (35,30)-(766,531): text "Sort short addresses"
rectangle at (85,190)-(116,221): text "1"; invisible if not DALI_Config.Kurzadr[1]; alarm colour if DALI_Config.mAlteAdresse[1]; toggles DALI_Config.AlteAdresse[1]
rectangle at (125,190)-(156,221): text "2"; invisible if not DALI_Config.Kurzadr[2]; alarm colour if DALI_Config.mAlteAdresse[2]; toggles DALI_Config.AlteAdresse[2]
rectangle at (165,190)-(196,221): text "3"; invisible if not DALI_Config.Kurzadr[3]; alarm colour if DALI_Config.mAlteAdresse[3]; toggles DALI_Config.AlteAdresse[3]
rectangle at (205,190)-(236,221): text "4"; invisible if not DALI_Config.Kurzadr[4]; alarm colour if DALI_Config.mAlteAdresse[4]; toggles DALI_Config.AlteAdresse[4]
rectangle at (245,190)-(276,221): text "5"; invisible if not DALI_Config.Kurzadr[5]; alarm colour if DALI_Config.mAlteAdresse[5]; toggles DALI_Config.AlteAdresse[5]
rectangle at (285,190)-(316,221): text "6"; invisible if not DALI_Config.Kurzadr[6]; alarm colour if DALI_Config.mAlteAdresse[6]; toggles DALI_Config.AlteAdresse[6]
rectangle at (325,190)-(356,221): text "7"; invisible if not DALI_Config.Kurzadr[7]; alarm colour if DALI_Config.mAlteAdresse[7]; toggles DALI_Config.AlteAdresse[7]
rectangle at (365,190)-(396,221): text "8"; invisible if not DALI_Config.Kurzadr[8]; alarm colour if DALI_Config.mAlteAdresse[8]; toggles DALI_Config.AlteAdresse[8]
rectangle at (405,190)-(436,221): text "9"; invisible if not DALI_Config.Kurzadr[9]; alarm colour if DALI_Config.mAlteAdresse[9]; toggles DALI_Config.AlteAdresse[9]
rectangle at (445,190)-(476,221): text "10"; invisible if not DALI_Config.Kurzadr[10]; alarm colour if DALI_Config.mAlteAdresse[10]; toggles DALI_Config.AlteAdresse[10]
rectangle at (485,190)-(516,221): text "11"; invisible if not DALI_Config.Kurzadr[11]; alarm colour if DALI_Config.mAlteAdresse[11]; toggles DALI_Config.AlteAdresse[11]
rectangle at (525,190)-(556,221): text "12"; invisible if not DALI_Config.Kurzadr[12]; alarm colour if DALI_Config.mAlteAdresse[12]; toggles DALI_Config.AlteAdresse[12]
rectangle at (565,190)-(596,221): text "13"; invisible if not DALI_Config.Kurzadr[13]; alarm colour if DALI_Config.mAlteAdresse[13]; toggles DALI_Config.AlteAdresse[13]
rectangle at (605,190)-(636,221): text "14"; invisible if not DALI_Config.Kurzadr[14]; alarm colour if DALI_Config.mAlteAdresse[14]; toggles DALI_Config.AlteAdresse[14]
rectangle at (645,190)-(676,221): text "15"; invisible if not DALI_Config.Kurzadr[15]; alarm colour if DALI_Config.mAlteAdresse[15]; toggles DALI_Config.AlteAdresse[15]
rectangle at (685,190)-(716,221): text "16"; invisible if not DALI_Config.Kurzadr[16]; alarm colour if DALI_Config.mAlteAdresse[16]; toggles DALI_Config.AlteAdresse[16]
rectangle at (85,230)-(116,261): text "17"; invisible if not DALI_Config.Kurzadr[17]; alarm colour if DALI_Config.mAlteAdresse[17]; toggles DALI_Config.AlteAdresse[17]
rectangle at (165,230)-(196,261): text "19"; invisible if not DALI_Config.Kurzadr[19]; alarm colour if DALI_Config.mAlteAdresse[19]; toggles DALI_Config.AlteAdresse[19]
rectangle at (125,230)-(156,261): text "18"; invisible if not DALI_Config.Kurzadr[18]; alarm colour if DALI_Config.mAlteAdresse[18]; toggles DALI_Config.AlteAdresse[18]
rectangle at (205,230)-(236,261): text "20"; invisible if not DALI_Config.Kurzadr[20]; alarm colour if DALI_Config.mAlteAdresse[20]; toggles DALI_Config.AlteAdresse[20]
rectangle at (245,230)-(276,261): text "21"; invisible if not DALI_Config.Kurzadr[21]; alarm colour if DALI_Config.mAlteAdresse[21]; toggles DALI_Config.AlteAdresse[21]
rectangle at (285,230)-(316,261): text "22"; invisible if not DALI_Config.Kurzadr[22]; alarm colour if DALI_Config.mAlteAdresse[22]; toggles DALI_Config.AlteAdresse[22]
rectangle at (325,230)-(356,261): text "23"; invisible if not DALI_Config.Kurzadr[23]; alarm colour if DALI_Config.mAlteAdresse[23]; toggles DALI_Config.AlteAdresse[23]
rectangle at (365,230)-(396,261): text "24"; invisible if not DALI_Config.Kurzadr[24]; alarm colour if DALI_Config.mAlteAdresse[24]; toggles DALI_Config.AlteAdresse[24]
rectangle at (405,230)-(436,261): text "25"; invisible if not DALI_Config.Kurzadr[25]; alarm colour if DALI_Config.mAlteAdresse[25]; toggles DALI_Config.AlteAdresse[25]
rectangle at (565,230)-(596,261): text "29"; invisible if not DALI_Config.Kurzadr[29]; alarm colour if DALI_Config.mAlteAdresse[29]; toggles DALI_Config.AlteAdresse[29]
rectangle at (525,230)-(556,261): text "28"; invisible if not DALI_Config.Kurzadr[28]; alarm colour if DALI_Config.mAlteAdresse[28]; toggles DALI_Config.AlteAdresse[28]
rectangle at (485,230)-(516,261): text "27"; invisible if not DALI_Config.Kurzadr[27]; alarm colour if DALI_Config.mAlteAdresse[27]; toggles DALI_Config.AlteAdresse[27]
rectangle at (445,230)-(476,261): text "26"; invisible if not DALI_Config.Kurzadr[26]; alarm colour if DALI_Config.mAlteAdresse[26]; toggles DALI_Config.AlteAdresse[26]
rectangle at (605,230)-(636,261): text "30"; invisible if not DALI_Config.Kurzadr[30]; alarm colour if DALI_Config.mAlteAdresse[30]; toggles DALI_Config.AlteAdresse[30]
rectangle at (645,230)-(676,261): text "31"; invisible if not DALI_Config.Kurzadr[31]; alarm colour if DALI_Config.mAlteAdresse[31]; toggles DALI_Config.AlteAdresse[31]
rectangle at (685,230)-(716,261): text "32"; invisible if not DALI_Config.Kurzadr[32]; alarm colour if DALI_Config.mAlteAdresse[32]; toggles DALI_Config.AlteAdresse[32]
rectangle at (85,270)-(116,301): text "33"; invisible if not DALI_Config.Kurzadr[33]; alarm colour if DALI_Config.mAlteAdresse[33]; toggles DALI_Config.AlteAdresse[33]
rectangle at (125,270)-(156,301): text "34"; invisible if not DALI_Config.Kurzadr[34]; alarm colour if DALI_Config.mAlteAdresse[34]; toggles DALI_Config.AlteAdresse[34]
rectangle at (205,270)-(236,301): text "36"; invisible if not DALI_Config.Kurzadr[36]; alarm colour if DALI_Config.mAlteAdresse[36]; toggles DALI_Config.AlteAdresse[36]
rectangle at (285,270)-(316,301): text "38"; invisible if not DALI_Config.Kurzadr[38]; alarm colour if DALI_Config.mAlteAdresse[38]; toggles DALI_Config.AlteAdresse[38]
rectangle at (325,270)-(356,301): text "39"; invisible if not DALI_Config.Kurzadr[39]; alarm colour if DALI_Config.mAlteAdresse[39]; toggles DALI_Config.AlteAdresse[39]
rectangle at (245,270)-(276,301): text "37"; invisible if not DALI_Config.Kurzadr[37]; alarm colour if DALI_Config.mAlteAdresse[37]; toggles DALI_Config.AlteAdresse[37]
rectangle at (165,270)-(196,301): text "35"; invisible if not DALI_Config.Kurzadr[35]; alarm colour if DALI_Config.mAlteAdresse[35]; toggles DALI_Config.AlteAdresse[35]
rectangle at (405,270)-(436,301): text "41"; invisible if not DALI_Config.Kurzadr[41]; alarm colour if DALI_Config.mAlteAdresse[41]; toggles DALI_Config.AlteAdresse[41]
rectangle at (445,270)-(476,301): text "42"; invisible if not DALI_Config.Kurzadr[42]; alarm colour if DALI_Config.mAlteAdresse[42]; toggles DALI_Config.AlteAdresse[42]
rectangle at (365,270)-(396,301): text "40"; invisible if not DALI_Config.Kurzadr[40]; alarm colour if DALI_Config.mAlteAdresse[40]; toggles DALI_Config.AlteAdresse[40]
rectangle at (485,270)-(516,301): text "43"; invisible if not DALI_Config.Kurzadr[43]; alarm colour if DALI_Config.mAlteAdresse[43]; toggles DALI_Config.AlteAdresse[43]
rectangle at (525,270)-(556,301): text "44"; invisible if not DALI_Config.Kurzadr[44]; alarm colour if DALI_Config.mAlteAdresse[44]; toggles DALI_Config.AlteAdresse[44]
rectangle at (565,270)-(596,301): text "45"; invisible if not DALI_Config.Kurzadr[45]; alarm colour if DALI_Config.mAlteAdresse[45]; toggles DALI_Config.AlteAdresse[45]
rectangle at (605,270)-(636,301): text "46"; invisible if not DALI_Config.Kurzadr[46]; alarm colour if DALI_Config.mAlteAdresse[46]; toggles DALI_Config.AlteAdresse[46]
rectangle at (645,270)-(676,301): text "47"; invisible if not DALI_Config.Kurzadr[47]; alarm colour if DALI_Config.mAlteAdresse[47]; toggles DALI_Config.AlteAdresse[47]
rectangle at (685,270)-(716,301): text "48"; invisible if not DALI_Config.Kurzadr[48]; alarm colour if DALI_Config.mAlteAdresse[48]; toggles DALI_Config.AlteAdresse[48]
rectangle at (85,310)-(116,341): text "49"; invisible if not DALI_Config.Kurzadr[49]; alarm colour if DALI_Config.mAlteAdresse[49]; toggles DALI_Config.AlteAdresse[49]
rectangle at (125,310)-(156,341): text "50"; invisible if not DALI_Config.Kurzadr[50]; alarm colour if DALI_Config.mAlteAdresse[50]; toggles DALI_Config.AlteAdresse[50]
rectangle at (165,310)-(196,341): text "51"; invisible if not DALI_Config.Kurzadr[51]; alarm colour if DALI_Config.mAlteAdresse[51]; toggles DALI_Config.AlteAdresse[51]
rectangle at (205,310)-(236,341): text "52"; invisible if not DALI_Config.Kurzadr[52]; alarm colour if DALI_Config.mAlteAdresse[52]; toggles DALI_Config.AlteAdresse[52]
rectangle at (245,310)-(276,341): text "53"; invisible if not DALI_Config.Kurzadr[53]; alarm colour if DALI_Config.mAlteAdresse[53]; toggles DALI_Config.AlteAdresse[53]
rectangle at (285,310)-(316,341): text "54"; invisible if not DALI_Config.Kurzadr[54]; alarm colour if DALI_Config.mAlteAdresse[54]; toggles DALI_Config.AlteAdresse[54]
rectangle at (325,310)-(356,341): text "55"; invisible if not DALI_Config.Kurzadr[55]; alarm colour if DALI_Config.mAlteAdresse[55]; toggles DALI_Config.AlteAdresse[55]
rectangle at (365,310)-(396,341): text "56"; invisible if not DALI_Config.Kurzadr[56]; alarm colour if DALI_Config.mAlteAdresse[56]; toggles DALI_Config.AlteAdresse[56]
rectangle at (405,310)-(436,341): text "57"; invisible if not DALI_Config.Kurzadr[57]; alarm colour if DALI_Config.mAlteAdresse[57]; toggles DALI_Config.AlteAdresse[57]
rectangle at (485,310)-(516,341): text "59"; invisible if not DALI_Config.Kurzadr[59]; alarm colour if DALI_Config.mAlteAdresse[59]; toggles DALI_Config.AlteAdresse[59]
rectangle at (525,310)-(556,341): text "60"; invisible if not DALI_Config.Kurzadr[60]; alarm colour if DALI_Config.mAlteAdresse[60]; toggles DALI_Config.AlteAdresse[60]
rectangle at (565,310)-(596,341): text "61"; invisible if not DALI_Config.Kurzadr[61]; alarm colour if DALI_Config.mAlteAdresse[61]; toggles DALI_Config.AlteAdresse[61]
rectangle at (605,310)-(636,341): text "62"; invisible if not DALI_Config.Kurzadr[62]; alarm colour if DALI_Config.mAlteAdresse[62]; toggles DALI_Config.AlteAdresse[62]
rectangle at (445,310)-(476,341): text "58"; invisible if not DALI_Config.Kurzadr[58]; alarm colour if DALI_Config.mAlteAdresse[58]; toggles DALI_Config.AlteAdresse[58]
rectangle at (645,310)-(676,341): text "63"; invisible if not DALI_Config.Kurzadr[63]; alarm colour if DALI_Config.mAlteAdresse[63]; toggles DALI_Config.AlteAdresse[63]
rectangle at (685,310)-(716,341): text "64"; invisible if not DALI_Config.Kurzadr[64]; alarm colour if DALI_Config.mAlteAdresse[64]; toggles DALI_Config.AlteAdresse[64]
rectangle at (85,190)-(116,221): text "1"; invisible if DALI_Config.Kurzadr[1]; alarm colour if DALI_Config.mNeueAdresse[1]; toggles DALI_Config.NeueAdresse[1]
rectangle at (125,190)-(156,221): text "2"; invisible if DALI_Config.Kurzadr[2]; alarm colour if DALI_Config.mNeueAdresse[2]; toggles DALI_Config.NeueAdresse[2]
rectangle at (405,190)-(436,221): text "9"; invisible if DALI_Config.Kurzadr[9]; alarm colour if DALI_Config.mNeueAdresse[9]; toggles DALI_Config.NeueAdresse[9]
rectangle at (165,190)-(196,221): text "3"; invisible if DALI_Config.Kurzadr[3]; alarm colour if DALI_Config.mNeueAdresse[3]; toggles DALI_Config.NeueAdresse[3]
rectangle at (205,190)-(236,221): text "4"; invisible if DALI_Config.Kurzadr[4]; alarm colour if DALI_Config.mNeueAdresse[4]; toggles DALI_Config.NeueAdresse[4]
rectangle at (245,190)-(276,221): text "5"; invisible if DALI_Config.Kurzadr[5]; alarm colour if DALI_Config.mNeueAdresse[5]; toggles DALI_Config.NeueAdresse[5]
rectangle at (285,190)-(316,221): text "6"; invisible if DALI_Config.Kurzadr[6]; alarm colour if DALI_Config.mNeueAdresse[6]; toggles DALI_Config.NeueAdresse[6]
rectangle at (325,190)-(356,221): text "7"; invisible if DALI_Config.Kurzadr[7]; alarm colour if DALI_Config.mNeueAdresse[7]; toggles DALI_Config.NeueAdresse[7]
rectangle at (365,190)-(396,221): text "8"; invisible if DALI_Config.Kurzadr[8]; alarm colour if DALI_Config.mNeueAdresse[8]; toggles DALI_Config.NeueAdresse[8]
rectangle at (445,190)-(476,221): text "10"; invisible if DALI_Config.Kurzadr[10]; alarm colour if DALI_Config.mNeueAdresse[10]; toggles DALI_Config.NeueAdresse[10]
rectangle at (485,190)-(516,221): text "11"; invisible if DALI_Config.Kurzadr[11]; alarm colour if DALI_Config.mNeueAdresse[11]; toggles DALI_Config.NeueAdresse[11]
rectangle at (525,190)-(556,221): text "12"; invisible if DALI_Config.Kurzadr[12]; alarm colour if DALI_Config.mNeueAdresse[12]; toggles DALI_Config.NeueAdresse[12]
rectangle at (565,190)-(596,221): text "13"; invisible if DALI_Config.Kurzadr[13]; alarm colour if DALI_Config.mNeueAdresse[13]; toggles DALI_Config.NeueAdresse[13]
rectangle at (605,190)-(636,221): text "14"; invisible if DALI_Config.Kurzadr[14]; alarm colour if DALI_Config.mNeueAdresse[14]; toggles DALI_Config.NeueAdresse[14]
rectangle at (645,190)-(676,221): text "15"; invisible if DALI_Config.Kurzadr[15]; alarm colour if DALI_Config.mNeueAdresse[15]; toggles DALI_Config.NeueAdresse[15]
rectangle at (85,230)-(116,261): text "17"; invisible if DALI_Config.Kurzadr[17]; alarm colour if DALI_Config.mNeueAdresse[17]; toggles DALI_Config.NeueAdresse[17]
rectangle at (125,230)-(156,261): text "18"; invisible if DALI_Config.Kurzadr[18]; alarm colour if DALI_Config.mNeueAdresse[18]; toggles DALI_Config.NeueAdresse[18]
rectangle at (685,190)-(716,221): text "16"; invisible if DALI_Config.Kurzadr[16]; alarm colour if DALI_Config.mNeueAdresse[16]; toggles DALI_Config.NeueAdresse[16]
rectangle at (405,230)-(436,261): text "25"; invisible if DALI_Config.Kurzadr[25]; alarm colour if DALI_Config.mNeueAdresse[25]; toggles DALI_Config.NeueAdresse[25]
rectangle at (165,230)-(196,261): text "19"; invisible if DALI_Config.Kurzadr[19]; alarm colour if DALI_Config.mNeueAdresse[19]; toggles DALI_Config.NeueAdresse[19]
rectangle at (205,230)-(236,261): text "20"; invisible if DALI_Config.Kurzadr[20]; alarm colour if DALI_Config.mNeueAdresse[20]; toggles DALI_Config.NeueAdresse[20]
rectangle at (285,230)-(316,261): text "22"; invisible if DALI_Config.Kurzadr[22]; alarm colour if DALI_Config.mNeueAdresse[22]; toggles DALI_Config.NeueAdresse[22]
rectangle at (325,230)-(356,261): text "23"; invisible if DALI_Config.Kurzadr[23]; alarm colour if DALI_Config.mNeueAdresse[23]; toggles DALI_Config.NeueAdresse[23]
rectangle at (245,230)-(276,261): text "21"; invisible if DALI_Config.Kurzadr[21]; alarm colour if DALI_Config.mNeueAdresse[21]; toggles DALI_Config.NeueAdresse[21]
rectangle at (365,230)-(396,261): text "24"; invisible if DALI_Config.Kurzadr[24]; alarm colour if DALI_Config.mNeueAdresse[24]; toggles DALI_Config.NeueAdresse[24]
rectangle at (445,230)-(476,261): text "26"; invisible if DALI_Config.Kurzadr[26]; alarm colour if DALI_Config.mNeueAdresse[26]; toggles DALI_Config.NeueAdresse[26]
rectangle at (485,230)-(516,261): text "27"; invisible if DALI_Config.Kurzadr[27]; alarm colour if DALI_Config.mNeueAdresse[27]; toggles DALI_Config.NeueAdresse[27]
rectangle at (525,230)-(556,261): text "28"; invisible if DALI_Config.Kurzadr[28]; alarm colour if DALI_Config.mNeueAdresse[28]; toggles DALI_Config.NeueAdresse[28]
rectangle at (645,230)-(676,261): text "31"; invisible if DALI_Config.Kurzadr[31]; alarm colour if DALI_Config.mNeueAdresse[31]; toggles DALI_Config.NeueAdresse[31]
rectangle at (565,230)-(596,261): text "29"; invisible if DALI_Config.Kurzadr[29]; alarm colour if DALI_Config.mNeueAdresse[29]; toggles DALI_Config.NeueAdresse[29]
rectangle at (685,230)-(716,261): text "32"; invisible if DALI_Config.Kurzadr[32]; alarm colour if DALI_Config.mNeueAdresse[32]; toggles DALI_Config.NeueAdresse[32]
rectangle at (85,270)-(116,301): text "33"; invisible if DALI_Config.Kurzadr[33]; alarm colour if DALI_Config.mNeueAdresse[33]; toggles DALI_Config.NeueAdresse[33]
rectangle at (125,270)-(156,301): text "34"; invisible if DALI_Config.Kurzadr[34]; alarm colour if DALI_Config.mNeueAdresse[34]; toggles DALI_Config.NeueAdresse[34]
rectangle at (605,230)-(636,261): text "30"; invisible if DALI_Config.Kurzadr[30]; alarm colour if DALI_Config.mNeueAdresse[30]; toggles DALI_Config.NeueAdresse[30]
rectangle at (165,270)-(196,301): text "35"; invisible if DALI_Config.Kurzadr[35]; alarm colour if DALI_Config.mNeueAdresse[35]; toggles DALI_Config.NeueAdresse[35]
rectangle at (205,270)-(236,301): text "36"; invisible if DALI_Config.Kurzadr[36]; alarm colour if DALI_Config.mNeueAdresse[36]; toggles DALI_Config.NeueAdresse[36]
rectangle at (245,270)-(276,301): text "37"; invisible if DALI_Config.Kurzadr[37]; alarm colour if DALI_Config.mNeueAdresse[37]; toggles DALI_Config.NeueAdresse[37]
rectangle at (285,270)-(316,301): text "38"; invisible if DALI_Config.Kurzadr[38]; alarm colour if DALI_Config.mNeueAdresse[38]; toggles DALI_Config.NeueAdresse[38]
rectangle at (325,270)-(356,301): text "39"; invisible if DALI_Config.Kurzadr[39]; alarm colour if DALI_Config.mNeueAdresse[39]; toggles DALI_Config.NeueAdresse[39]
rectangle at (525,270)-(556,301): text "44"; invisible if DALI_Config.Kurzadr[44]; alarm colour if DALI_Config.mNeueAdresse[44]; toggles DALI_Config.NeueAdresse[44]
rectangle at (485,270)-(516,301): text "43"; invisible if DALI_Config.Kurzadr[43]; alarm colour if DALI_Config.mNeueAdresse[43]; toggles DALI_Config.NeueAdresse[43]
rectangle at (445,270)-(476,301): text "42"; invisible if DALI_Config.Kurzadr[42]; alarm colour if DALI_Config.mNeueAdresse[42]; toggles DALI_Config.NeueAdresse[42]
rectangle at (405,270)-(436,301): text "41"; invisible if DALI_Config.Kurzadr[41]; alarm colour if DALI_Config.mNeueAdresse[41]; toggles DALI_Config.NeueAdresse[41]
rectangle at (365,270)-(396,301): text "40"; invisible if DALI_Config.Kurzadr[40]; alarm colour if DALI_Config.mNeueAdresse[40]; toggles DALI_Config.NeueAdresse[40]
rectangle at (565,270)-(596,301): text "45"; invisible if DALI_Config.Kurzadr[45]; alarm colour if DALI_Config.mNeueAdresse[45]; toggles DALI_Config.NeueAdresse[45]
rectangle at (605,270)-(636,301): text "46"; invisible if DALI_Config.Kurzadr[46]; alarm colour if DALI_Config.mNeueAdresse[46]; toggles DALI_Config.NeueAdresse[46]
rectangle at (645,270)-(676,301): text "47"; invisible if DALI_Config.Kurzadr[47]; alarm colour if DALI_Config.mNeueAdresse[47]; toggles DALI_Config.NeueAdresse[47]
rectangle at (685,270)-(716,301): text "48"; invisible if DALI_Config.Kurzadr[48]; alarm colour if DALI_Config.mNeueAdresse[48]; toggles DALI_Config.NeueAdresse[48]
rectangle at (85,310)-(116,341): text "49"; invisible if DALI_Config.Kurzadr[49]; alarm colour if DALI_Config.mNeueAdresse[49]; toggles DALI_Config.NeueAdresse[49]
rectangle at (125,310)-(156,341): text "50"; invisible if DALI_Config.Kurzadr[50]; alarm colour if DALI_Config.mNeueAdresse[50]; toggles DALI_Config.NeueAdresse[50]
rectangle at (165,310)-(196,341): text "51"; invisible if DALI_Config.Kurzadr[51]; alarm colour if DALI_Config.mNeueAdresse[51]; toggles DALI_Config.NeueAdresse[51]
rectangle at (205,310)-(236,341): text "52"; invisible if DALI_Config.Kurzadr[52]; alarm colour if DALI_Config.mNeueAdresse[52]; toggles DALI_Config.NeueAdresse[52]
rectangle at (245,310)-(276,341): text "53"; invisible if DALI_Config.Kurzadr[53]; alarm colour if DALI_Config.mNeueAdresse[53]; toggles DALI_Config.NeueAdresse[53]
rectangle at (325,310)-(356,341): text "55"; invisible if DALI_Config.Kurzadr[55]; alarm colour if DALI_Config.mNeueAdresse[55]; toggles DALI_Config.NeueAdresse[55]
rectangle at (405,310)-(436,341): text "57"; invisible if DALI_Config.Kurzadr[57]; alarm colour if DALI_Config.mNeueAdresse[57]; toggles DALI_Config.NeueAdresse[57]
rectangle at (445,310)-(476,341): text "58"; invisible if DALI_Config.Kurzadr[58]; alarm colour if DALI_Config.mNeueAdresse[58]; toggles DALI_Config.NeueAdresse[58]
rectangle at (365,310)-(396,341): text "56"; invisible if DALI_Config.Kurzadr[56]; alarm colour if DALI_Config.mNeueAdresse[56]; toggles DALI_Config.NeueAdresse[56]
rectangle at (285,310)-(316,341): text "54"; invisible if DALI_Config.Kurzadr[54]; alarm colour if DALI_Config.mNeueAdresse[54]; toggles DALI_Config.NeueAdresse[54]
rectangle at (485,310)-(516,341): text "59"; invisible if DALI_Config.Kurzadr[59]; alarm colour if DALI_Config.mNeueAdresse[59]; toggles DALI_Config.NeueAdresse[59]
rectangle at (525,310)-(556,341): text "60"; invisible if DALI_Config.Kurzadr[60]; alarm colour if DALI_Config.mNeueAdresse[60]; toggles DALI_Config.NeueAdresse[60]
rectangle at (565,310)-(596,341): text "61"; invisible if DALI_Config.Kurzadr[61]; alarm colour if DALI_Config.mNeueAdresse[61]; toggles DALI_Config.NeueAdresse[61]
rectangle at (685,310)-(716,341): text "64"; invisible if DALI_Config.Kurzadr[64]; alarm colour if DALI_Config.mNeueAdresse[64]; toggles DALI_Config.NeueAdresse[64]
rectangle at (605,310)-(636,341): text "62"; invisible if DALI_Config.Kurzadr[62]; alarm colour if DALI_Config.mNeueAdresse[62]; toggles DALI_Config.NeueAdresse[62]
rectangle at (645,310)-(676,341): text "63"; invisible if DALI_Config.Kurzadr[63]; alarm colour if DALI_Config.mNeueAdresse[63]; toggles DALI_Config.NeueAdresse[63]
button at (325,125)-(471,161): text "Change"; taps DALI_Config.Tausch; tooltip If you click the button "Change", the old short address will be replaced by the new short address.
button at (590,370)-(736,406): text "Blink"; taps DALI_Config.xBlinken; tooltip If you click the button "Blink", the selected ECG will blink as long as defined by the "Blink Time" parameter.
button at (590,420)-(736,456): text "Stop blinking"; taps DALI_Config.xBlinken_Aus; tooltip If you click the button "Stop blinking", the blinking of the ECG will stop immediately.
rectangle at (90,380)-(251,401): text "Short address available"
rectangle at (100,410)-(231,431): text "Old short address"
rectangle at (105,440)-(236,461): text "New short address"
rounded rectangle at (330,470)-(476,506): text "Home page"; opens DALI; tooltip Back to home page
rectangle at (590,470)-(696,506): text "Blink time [sek]"
rectangle at (700,470)-(736,506): text "%s"; shows DALI_Config.bBlinkzeit; tooltip Enter blink time (3 - 255 seconds); editable
button at (330,370)-(476,406): text "Central On"; taps DALI_Config.Ein; tooltip If you click the button "Central On", all lamps in the network will be switched on.
button at (330,420)-(476,456): text "Central Off"; taps DALI_Config.Aus; tooltip If you click the button "Central Off", all lamps in the network will be switched off.
rounded rectangle at (130,75)-(666,111): text "DALI Line %s"; shows DALI_Config.bDali_Linie; tooltip You can change the DALI Line only on the home page.
6 more shapes without text or variables
*)

(* Visualisation Visualizace
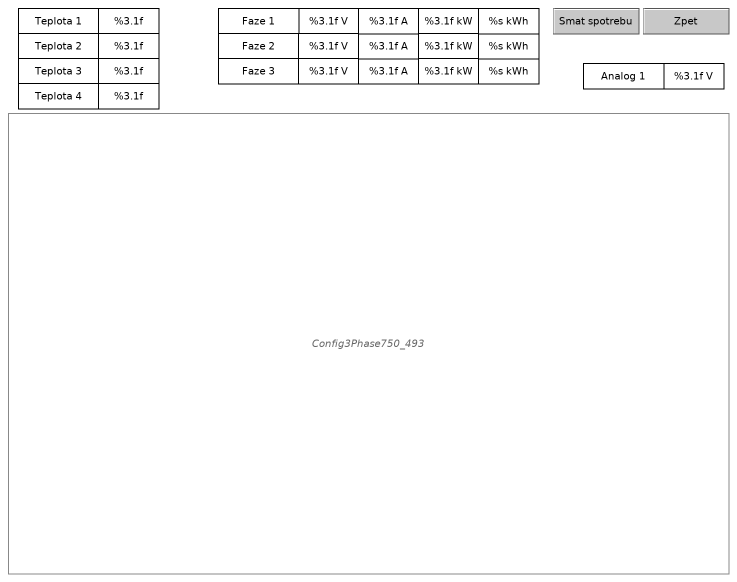
rectangle at (30,35)-(111,61): text "Teplota 1"
rectangle at (30,60)-(111,86): text "Teplota 2"
rectangle at (30,85)-(111,111): text "Teplota 3"
rectangle at (30,110)-(111,136): text "Teplota 4"
rectangle at (110,35)-(171,61): text "%3.1f"; shows .Teplota_1/10.0
rectangle at (110,60)-(171,86): text "%3.1f"; shows .Teplota_2/10.0
rectangle at (110,85)-(171,111): text "%3.1f"; shows .Teplota_3/10.0
rectangle at (110,110)-(171,136): text "%3.1f"; shows .Teplota_4/10.0
rectangle at (675,90)-(736,116): text "%3.1f V"; shows .Analog_1/3276.4
rectangle at (595,90)-(676,116): text "Analog 1"
rectangle at (310,35)-(371,61): text "%3.1f V"; shows TriFaze.arNapeti[1]
rectangle at (230,35)-(311,61): text "Faze 1"
rectangle at (230,60)-(311,86): text "Faze 2"
rectangle at (230,85)-(311,111): text "Faze 3"
embedded screen at (20,140)-(741,601): Config3Phase750_493
rectangle at (310,60)-(371,86): text "%3.1f V"; shows TriFaze.arNapeti[2]
rectangle at (310,85)-(371,111): text "%3.1f V"; shows TriFaze.arNapeti[3]
rectangle at (370,85)-(431,111): text "%3.1f A"; shows TriFaze.arProud[3]
rectangle at (370,60)-(431,86): text "%3.1f A"; shows TriFaze.arProud[2]
rectangle at (370,35)-(431,61): text "%3.1f A"; shows TriFaze.arProud[1]
rectangle at (430,35)-(491,61): text "%3.1f kW"; shows TriFaze.arVykon[1]
rectangle at (430,60)-(491,86): text "%3.1f kW"; shows TriFaze.arVykon[2]
rectangle at (430,85)-(491,111): text "%3.1f kW"; shows TriFaze.arVykon[3]
rectangle at (490,85)-(551,111): text "%s kWh"; shows TriFaze.adwSpotreba[3]
rectangle at (490,60)-(551,86): text "%s kWh"; shows TriFaze.adwSpotreba[2]
rectangle at (490,35)-(551,61): text "%s kWh"; shows TriFaze.adwSpotreba[1]
button at (565,35)-(651,61): text "Smat spotrebu"; taps TriFaze.SmazL1
button at (655,35)-(741,61): text "Zpet"; opens PLC_VISU
*)
